LIN {X 98.42, Y 171.93, Z 0.00, A 0, B 0, C 0} C_DIS
LIN {X 98.57, Y 172.17, Z 0.00, A 0, B 0, C 0} C_DIS
LIN {X 98.70, Y 172.42, Z 0.00, A 0, B 0, C 0} C_DIS
LIN {X 98.83, Y 172.69, Z 0.00, A 0, B 0, C 0} C_DIS
LIN {X 98.95, Y 172.96, Z 0.00, A 0, B 0, C 0} C_DIS
LIN {X 99.07, Y 173.23, Z 0.00, A 0, B 0, C 0} C_DIS
LIN {X 99.19, Y 173.50, Z 0.00, A 0, B 0, C 0} C_DIS
LIN {X 99.31, Y 173.78, Z 0.00, A 0, B 0, C 0} C_DIS
LIN {X 99.43, Y 174.05, Z 0.00, A 0, B 0, C 0} C_DIS
LIN {X 99.55, Y 174.33, Z 0.00, A 0, B 0, C 0} C_DIS
LIN {X 99.67, Y 174.60, Z 0.00, A 0, B 0, C 0} C_DIS
LIN {X 99.79, Y 174.87, Z 0.00, A 0, B 0, C 0} C_DIS
LIN {X 99.92, Y 175.14, Z 0.00, A 0, B 0, C 0} C_DIS
LIN {X 100.03, Y 175.42, Z 0.00, A 0, B 0, C 0} C_DIS
LIN {X 100.12, Y 175.71, Z 0.00, A 0, B 0, C 0} C_DIS
LIN {X 100.21, Y 176.02, Z 0.00, A 0, B 0, C 0} C_DIS
LIN {X 100.30, Y 176.31, Z 0.00, A 0, B 0, C 0} C_DIS
LIN {X 100.41, Y 176.59, Z 0.00, A 0, B 0, C 0} C_DIS
LIN {X 100.52, Y 176.87, Z 0.00, A 0, B 0, C 0} C_DIS
LIN {X 100.64, Y 177.14, Z 0.00, A 0, B 0, C 0} C_DIS
LIN {X 100.77, Y 177.41, Z 0.00, A 0, B 0, C 0} C_DIS
LIN {X 100.89, Y 177.68, Z 0.00, A 0, B 0, C 0} C_DIS
LIN {X 101.02, Y 177.95, Z 0.00, A 0, B 0, C 0} C_DIS
LIN {X 101.14, Y 178.22, Z 0.00, A 0, B 0, C 0} C_DIS
LIN {X 101.26, Y 178.50, Z 0.00, A 0, B 0, C 0} C_DIS
LIN {X 101.36, Y 178.79, Z 0.00, A 0, B 0, C 0} C_DIS
LIN {X 101.45, Y 179.08, Z 0.00, A 0, B 0, C 0} C_DIS
LIN {X 101.54, Y 179.38, Z 0.00, A 0, B 0, C 0} C_DIS
LIN {X 101.64, Y 179.67, Z 0.00, A 0, B 0, C 0} C_DIS
LIN {X 101.75, Y 179.95, Z 0.00, A 0, B 0, C 0} C_DIS
LIN {X 101.85, Y 180.24, Z 0.00, A 0, B 0, C 0} C_DIS
LIN {X 101.93, Y 180.55, Z 0.00, A 0, B 0, C 0} C_DIS
LIN {X 102.02, Y 180.85, Z 0.00, A 0, B 0, C 0} C_DIS
LIN {X 102.12, Y 181.13, Z 0.00, A 0, B 0, C 0} C_DIS
LIN {X 102.23, Y 181.41, Z 0.00, A 0, B 0, C 0} C_DIS
LIN {X 102.33, Y 181.71, Z 0.00, A 0, B 0, C 0} C_DIS
LIN {X 102.41, Y 182.01, Z 0.00, A 0, B 0, C 0} C_DIS
LIN {X 102.51, Y 182.30, Z 0.00, A 0, B 0, C 0} C_DIS
LIN {X 102.61, Y 182.59, Z 0.00, A 0, B 0, C 0} C_DIS
LIN {X 102.72, Y 182.87, Z 0.00, A 0, B 0, C 0} C_DIS
LIN {X 102.81, Y 183.17, Z 0.00, A 0, B 0, C 0} C_DIS
LIN {X 102.89, Y 183.48, Z 0.00, A 0, B 0, C 0} C_DIS
LIN {X 103.00, Y 183.76, Z 0.00, A 0, B 0, C 0} C_DIS
LIN {X 103.12, Y 184.03, Z 0.00, A 0, B 0, C 0} C_DIS
LIN {X 103.20, Y 184.34, Z 0.00, A 0, B 0, C 0} C_DIS
LIN {X 103.25, Y 184.65, Z 0.00, A 0, B 0, C 0} C_DIS
LIN {X 103.31, Y 184.97, Z 0.00, A 0, B 0, C 0} C_DIS
LIN {X 103.40, Y 185.27, Z 0.00, A 0, B 0, C 0} C_DIS
LIN {X 103.49, Y 185.57, Z 0.00, A 0, B 0, C 0} C_DIS
LIN {X 103.57, Y 185.87, Z 0.00, A 0, B 0, C 0} C_DIS
LIN {X 103.62, Y 186.19, Z 0.00, A 0, B 0, C 0} C_DIS
LIN {X 103.67, Y 186.51, Z 0.00, A 0, B 0, C 0} C_DIS
LIN {X 103.72, Y 186.83, Z 0.00, A 0, B 0, C 0} C_DIS
LIN {X 103.80, Y 187.13, Z 0.00, A 0, B 0, C 0} C_DIS
LIN {X 103.89, Y 187.43, Z 0.00, A 0, B 0, C 0} C_DIS
LIN {X 103.98, Y 187.73, Z 0.00, A 0, B 0, C 0} C_DIS
LIN {X 104.04, Y 188.04, Z 0.00, A 0, B 0, C 0} C_DIS
LIN {X 104.09, Y 188.37, Z 0.00, A 0, B 0, C 0} C_DIS
LIN {X 104.13, Y 188.69, Z 0.00, A 0, B 0, C 0} C_DIS
LIN {X 104.21, Y 189.00, Z 0.00, A 0, B 0, C 0} C_DIS
LIN {X 104.30, Y 189.29, Z 0.00, A 0, B 0, C 0} C_DIS
LIN {X 104.38, Y 189.59, Z 0.00, A 0, B 0, C 0} C_DIS
LIN {X 104.45, Y 189.91, Z 0.00, A 0, B 0, C 0} C_DIS
LIN {X 104.51, Y 190.22, Z 0.00, A 0, B 0, C 0} C_DIS
LIN {X 104.56, Y 190.54, Z 0.00, A 0, B 0, C 0} C_DIS
LIN {X 104.62, Y 190.85, Z 0.00, A 0, B 0, C 0} C_DIS
LIN {X 104.70, Y 191.16, Z 0.00, A 0, B 0, C 0} C_DIS
LIN {X 104.78, Y 191.46, Z 0.00, A 0, B 0, C 0} C_DIS
LIN {X 104.86, Y 191.77, Z 0.00, A 0, B 0, C 0} C_DIS
LIN {X 104.93, Y 192.08, Z 0.00, A 0, B 0, C 0} C_DIS
LIN {X 104.99, Y 192.39, Z 0.00, A 0, B 0, C 0} C_DIS
LIN {X 105.04, Y 192.71, Z 0.00, A 0, B 0, C 0} C_DIS
LIN {X 105.08, Y 193.03, Z 0.00, A 0, B 0, C 0} C_DIS
LIN {X 105.13, Y 193.35, Z 0.00, A 0, B 0, C 0} C_DIS
LIN {X 105.18, Y 193.67, Z 0.00, A 0, B 0, C 0} C_DIS
LIN {X 105.23, Y 193.99, Z 0.00, A 0, B 0, C 0} C_DIS
LIN {X 105.29, Y 194.31, Z 0.00, A 0, B 0, C 0} C_DIS
LIN {X 105.35, Y 194.62, Z 0.00, A 0, B 0, C 0} C_DIS
LIN {X 105.41, Y 194.94, Z 0.00, A 0, B 0, C 0} C_DIS
LIN {X 105.46, Y 195.25, Z 0.00, A 0, B 0, C 0} C_DIS
LIN {X 105.50, Y 195.57, Z 0.00, A 0, B 0, C 0} C_DIS
LIN {X 105.54, Y 195.90, Z 0.00, A 0, B 0, C 0} C_DIS
LIN {X 105.58, Y 196.22, Z 0.00, A 0, B 0, C 0} C_DIS
LIN {X 105.61, Y 196.54, Z 0.00, A 0, B 0, C 0} C_DIS
LIN {X 105.64, Y 196.87, Z 0.00, A 0, B 0, C 0} C_DIS
LIN {X 105.67, Y 197.19, Z 0.00, A 0, B 0, C 0} C_DIS
LIN {X 105.71, Y 197.51, Z 0.00, A 0, B 0, C 0} C_DIS
LIN {X 105.76, Y 197.83, Z 0.00, A 0, B 0, C 0} C_DIS
LIN {X 105.82, Y 198.15, Z 0.00, A 0, B 0, C 0} C_DIS
LIN {X 105.88, Y 198.46, Z 0.00, A 0, B 0, C 0} C_DIS
LIN {X 105.93, Y 198.78, Z 0.00, A 0, B 0, C 0} C_DIS
LIN {X 105.98, Y 199.10, Z 0.00, A 0, B 0, C 0} C_DIS
LIN {X 106.02, Y 199.42, Z 0.00, A 0, B 0, C 0} C_DIS
LIN {X 106.04, Y 199.75, Z 0.00, A 0, B 0, C 0} C_DIS
LIN {X 106.04, Y 200.08, Z 0.00, A 0, B 0, C 0} C_DIS
LIN {X 106.04, Y 200.41, Z 0.00, A 0, B 0, C 0} C_DIS
LIN {X 106.03, Y 200.74, Z 0.00, A 0, B 0, C 0} C_DIS
LIN {X 106.03, Y 201.06, Z 0.00, A 0, B 0, C 0} C_DIS
LIN {X 106.05, Y 201.39, Z 0.00, A 0, B 0, C 0} C_DIS
LIN {X 106.09, Y 201.71, Z 0.00, A 0, B 0, C 0} C_DIS
LIN {X 106.13, Y 202.03, Z 0.00, A 0, B 0, C 0} C_DIS
LIN {X 106.19, Y 202.35, Z 0.00, A 0, B 0, C 0} C_DIS
LIN {X 106.25, Y 202.66, Z 0.00, A 0, B 0, C 0} C_DIS
LIN {X 106.30, Y 202.98, Z 0.00, A 0, B 0, C 0} C_DIS
LIN {X 106.36, Y 203.30, Z 0.00, A 0, B 0, C 0} C_DIS
LIN {X 106.40, Y 203.62, Z 0.00, A 0, B 0, C 0} C_DIS
LIN {X 106.43, Y 203.94, Z 0.00, A 0, B 0, C 0} C_DIS
LIN {X 106.46, Y 204.27, Z 0.00, A 0, B 0, C 0} C_DIS
LIN {X 106.48, Y 204.59, Z 0.00, A 0, B 0, C 0} C_DIS
LIN {X 106.48, Y 204.92, Z 0.00, A 0, B 0, C 0} C_DIS
LIN {X 106.48, Y 205.25, Z 0.00, A 0, B 0, C 0} C_DIS
LIN {X 106.47, Y 205.58, Z 0.00, A 0, B 0, C 0} C_DIS
LIN {X 106.46, Y 205.91, Z 0.00, A 0, B 0, C 0} C_DIS
LIN {X 106.46, Y 206.24, Z 0.00, A 0, B 0, C 0} C_DIS
LIN {X 106.48, Y 206.56, Z 0.00, A 0, B 0, C 0} C_DIS
LIN {X 106.52, Y 206.88, Z 0.00, A 0, B 0, C 0} C_DIS
LIN {X 106.56, Y 207.20, Z 0.00, A 0, B 0, C 0} C_DIS
LIN {X 106.61, Y 207.52, Z 0.00, A 0, B 0, C 0} C_DIS
LIN {X 106.66, Y 207.85, Z 0.00, A 0, B 0, C 0} C_DIS
LIN {X 106.73, Y 208.16, Z 0.00, A 0, B 0, C 0} C_DIS
LIN {X 106.83, Y 208.44, Z 0.00, A 0, B 0, C 0} C_DIS
LIN {X 106.96, Y 208.69, Z 0.00, A 0, B 0, C 0} C_DIS
LIN {X 107.12, Y 208.92, Z 0.00, A 0, B 0, C 0} C_DIS
LIN {X 107.28, Y 209.15, Z 0.00, A 0, B 0, C 0} C_DIS
LIN {X 107.43, Y 209.39, Z 0.00, A 0, B 0, C 0} C_DIS
LIN {X 107.60, Y 209.58, Z 0.00, A 0, B 0, C 0} C_DIS
LIN {X 107.80, Y 209.69, Z 0.00, A 0, B 0, C 0} C_DIS
LIN {X 108.02, Y 209.75, Z 0.00, A 0, B 0, C 0} C_DIS
LIN {X 108.24, Y 209.76, Z 0.00, A 0, B 0, C 0} C_DIS
LIN {X 108.46, Y 209.74, Z 0.00, A 0, B 0, C 0} C_DIS
LIN {X 108.67, Y 209.69, Z 0.00, A 0, B 0, C 0} C_DIS
LIN {X 108.89, Y 209.62, Z 0.00, A 0, B 0, C 0} C_DIS
LIN {X 109.10, Y 209.55, Z 0.00, A 0, B 0, C 0} C_DIS
LIN {X 109.31, Y 209.46, Z 0.00, A 0, B 0, C 0} C_DIS
LIN {X 109.52, Y 209.38, Z 0.00, A 0, B 0, C 0} C_DIS
LIN {X 109.73, Y 209.30, Z 0.00, A 0, B 0, C 0} C_DIS
LIN {X 109.94, Y 209.23, Z 0.00, A 0, B 0, C 0} C_DIS
LIN {X 110.15, Y 209.15, Z 0.00, A 0, B 0, C 0} C_DIS
LIN {X 110.36, Y 209.07, Z 0.00, A 0, B 0, C 0} C_DIS
LIN {X 110.57, Y 208.98, Z 0.00, A 0, B 0, C 0} C_DIS
LIN {X 110.78, Y 208.89, Z 0.00, A 0, B 0, C 0} C_DIS
LIN {X 111.00, Y 208.82, Z 0.00, A 0, B 0, C 0} C_DIS
LIN {X 111.21, Y 208.76, Z 0.00, A 0, B 0, C 0} C_DIS
LIN {X 111.42, Y 208.73, Z 0.00, A 0, B 0, C 0} C_DIS
LIN {X 111.64, Y 208.72, Z 0.00, A 0, B 0, C 0} C_DIS
LIN {X 111.86, Y 208.72, Z 0.00, A 0, B 0, C 0} C_DIS
LIN {X 112.08, Y 208.72, Z 0.00, A 0, B 0, C 0} C_DIS
LIN {X 112.29, Y 208.72, Z 0.00, A 0, B 0, C 0} C_DIS
LIN {X 112.51, Y 208.72, Z 0.00, A 0, B 0, C 0} C_DIS
LIN {X 112.73, Y 208.72, Z 0.00, A 0, B 0, C 0} C_DIS
LIN {X 112.95, Y 208.72, Z 0.00, A 0, B 0, C 0} C_DIS
LIN {X 113.16, Y 208.72, Z 0.00, A 0, B 0, C 0} C_DIS
LIN {X 113.38, Y 208.72, Z 0.00, A 0, B 0, C 0} C_DIS
LIN {X 113.60, Y 208.72, Z 0.00, A 0, B 0, C 0} C_DIS
LIN {X 113.82, Y 208.72, Z 0.00, A 0, B 0, C 0} C_DIS
LIN {X 114.03, Y 208.72, Z 0.00, A 0, B 0, C 0} C_DIS
LIN {X 114.25, Y 208.72, Z 0.00, A 0, B 0, C 0} C_DIS
LIN {X 114.47, Y 208.72, Z 0.00, A 0, B 0, C 0} C_DIS
LIN {X 114.69, Y 208.72, Z 0.00, A 0, B 0, C 0} C_DIS
LIN {X 114.90, Y 208.73, Z 0.00, A 0, B 0, C 0} C_DIS
LIN {X 115.12, Y 208.73, Z 0.00, A 0, B 0, C 0} C_DIS
LIN {X 115.34, Y 208.73, Z 0.00, A 0, B 0, C 0} C_DIS
LIN {X 115.56, Y 208.73, Z 0.00, A 0, B 0, C 0} C_DIS
LIN {X 115.77, Y 208.73, Z 0.00, A 0, B 0, C 0} C_DIS
LIN {X 115.99, Y 208.73, Z 0.00, A 0, B 0, C 0} C_DIS
LIN {X 116.21, Y 208.72, Z 0.00, A 0, B 0, C 0} C_DIS
LIN {X 116.43, Y 208.72, Z 0.00, A 0, B 0, C 0} C_DIS
LIN {X 116.64, Y 208.72, Z 0.00, A 0, B 0, C 0} C_DIS
LIN {X 116.86, Y 208.72, Z 0.00, A 0, B 0, C 0} C_DIS
LIN {X 117.08, Y 208.72, Z 0.00, A 0, B 0, C 0} C_DIS
LIN {X 117.30, Y 208.72, Z 0.00, A 0, B 0, C 0} C_DIS
LIN {X 117.51, Y 208.72, Z 0.00, A 0, B 0, C 0} C_DIS
LIN {X 117.73, Y 208.72, Z 0.00, A 0, B 0, C 0} C_DIS
LIN {X 117.95, Y 208.72, Z 0.00, A 0, B 0, C 0} C_DIS
LIN {X 118.17, Y 208.72, Z 0.00, A 0, B 0, C 0} C_DIS
LIN {X 118.38, Y 208.72, Z 0.00, A 0, B 0, C 0} C_DIS
LIN {X 118.60, Y 208.73, Z 0.00, A 0, B 0, C 0} C_DIS
LIN {X 118.82, Y 208.73, Z 0.00, A 0, B 0, C 0} C_DIS
LIN {X 119.04, Y 208.74, Z 0.00, A 0, B 0, C 0} C_DIS
LIN {X 119.25, Y 208.74, Z 0.00, A 0, B 0, C 0} C_DIS
LIN {X 119.47, Y 208.73, Z 0.00, A 0, B 0, C 0} C_DIS
LIN {X 119.69, Y 208.72, Z 0.00, A 0, B 0, C 0} C_DIS
LIN {X 119.90, Y 208.69, Z 0.00, A 0, B 0, C 0} C_DIS
LIN {X 120.12, Y 208.65, Z 0.00, A 0, B 0, C 0} C_DIS
LIN {X 120.33, Y 208.59, Z 0.00, A 0, B 0, C 0} C_DIS
LIN {X 120.55, Y 208.52, Z 0.00, A 0, B 0, C 0} C_DIS
LIN {X 120.76, Y 208.44, Z 0.00, A 0, B 0, C 0} C_DIS
LIN {X 120.96, Y 208.33, Z 0.00, A 0, B 0, C 0} C_DIS
LIN {X 121.16, Y 208.19, Z 0.00, A 0, B 0, C 0} C_DIS
LIN {X 121.32, Y 207.98, Z 0.00, A 0, B 0, C 0} C_DIS
LIN {X 121.47, Y 207.75, Z 0.00, A 0, B 0, C 0} C_DIS
LIN {X 121.64, Y 207.52, Z 0.00, A 0, B 0, C 0} C_DIS
LIN {X 121.78, Y 207.28, Z 0.00, A 0, B 0, C 0} C_DIS
LIN {X 121.90, Y 207.01, Z 0.00, A 0, B 0, C 0} C_DIS
LIN {X 121.99, Y 206.71, Z 0.00, A 0, B 0, C 0} C_DIS
LIN {X 122.06, Y 206.40, Z 0.00, A 0, B 0, C 0} C_DIS
LIN {X 122.11, Y 206.08, Z 0.00, A 0, B 0, C 0} C_DIS
LIN {X 122.15, Y 205.76, Z 0.00, A 0, B 0, C 0} C_DIS
LIN {X 122.17, Y 205.43, Z 0.00, A 0, B 0, C 0} C_DIS
LIN {X 122.20, Y 205.11, Z 0.00, A 0, B 0, C 0} C_DIS
LIN {X 122.21, Y 204.78, Z 0.00, A 0, B 0, C 0} C_DIS
LIN {X 122.22, Y 204.45, Z 0.00, A 0, B 0, C 0} C_DIS
LIN {X 122.22, Y 204.13, Z 0.00, A 0, B 0, C 0} C_DIS
LIN {X 122.22, Y 203.80, Z 0.00, A 0, B 0, C 0} C_DIS
LIN {X 122.22, Y 203.47, Z 0.00, A 0, B 0, C 0} C_DIS
LIN {X 122.22, Y 203.14, Z 0.00, A 0, B 0, C 0} C_DIS
LIN {X 122.22, Y 202.82, Z 0.00, A 0, B 0, C 0} C_DIS
LIN {X 122.21, Y 202.49, Z 0.00, A 0, B 0, C 0} C_DIS
LIN {X 122.21, Y 202.16, Z 0.00, A 0, B 0, C 0} C_DIS
LIN {X 122.21, Y 201.83, Z 0.00, A 0, B 0, C 0} C_DIS
LIN {X 122.21, Y 201.51, Z 0.00, A 0, B 0, C 0} C_DIS
LIN {X 122.21, Y 201.18, Z 0.00, A 0, B 0, C 0} C_DIS
LIN {X 122.21, Y 200.85, Z 0.00, A 0, B 0, C 0} C_DIS
LIN {X 122.21, Y 200.52, Z 0.00, A 0, B 0, C 0} C_DIS
LIN {X 122.22, Y 200.20, Z 0.00, A 0, B 0, C 0} C_DIS
LIN {X 122.22, Y 199.87, Z 0.00, A 0, B 0, C 0} C_DIS
LIN {X 122.22, Y 199.54, Z 0.00, A 0, B 0, C 0} C_DIS
LIN {X 122.22, Y 199.21, Z 0.00, A 0, B 0, C 0} C_DIS
LIN {X 122.22, Y 198.88, Z 0.00, A 0, B 0, C 0} C_DIS
LIN {X 122.22, Y 198.56, Z 0.00, A 0, B 0, C 0} C_DIS
LIN {X 122.20, Y 198.23, Z 0.00, A 0, B 0, C 0} C_DIS
LIN {X 122.20, Y 197.90, Z 0.00, A 0, B 0, C 0} C_DIS
LIN {X 122.21, Y 197.58, Z 0.00, A 0, B 0, C 0} C_DIS
LIN {X 122.25, Y 197.25, Z 0.00, A 0, B 0, C 0} C_DIS
LIN {X 122.34, Y 196.94, Z 0.00, A 0, B 0, C 0} C_DIS
LIN {X 122.46, Y 196.66, Z 0.00, A 0, B 0, C 0} C_DIS
LIN {X 122.62, Y 196.45, Z 0.00, A 0, B 0, C 0} C_DIS
LIN {X 122.82, Y 196.34, Z 0.00, A 0, B 0, C 0} C_DIS
LIN {X 123.03, Y 196.30, Z 0.00, A 0, B 0, C 0} C_DIS
LIN {X 123.25, Y 196.28, Z 0.00, A 0, B 0, C 0} C_DIS
LIN {X 123.47, Y 196.28, Z 0.00, A 0, B 0, C 0} C_DIS
LIN {X 123.69, Y 196.27, Z 0.00, A 0, B 0, C 0} C_DIS
LIN {X 123.91, Y 196.27, Z 0.00, A 0, B 0, C 0} C_DIS
LIN {X 124.13, Y 196.27, Z 0.00, A 0, B 0, C 0} C_DIS
LIN {X 124.35, Y 196.27, Z 0.00, A 0, B 0, C 0} C_DIS
LIN {X 124.56, Y 196.26, Z 0.00, A 0, B 0, C 0} C_DIS
LIN {X 124.78, Y 196.26, Z 0.00, A 0, B 0, C 0} C_DIS
LIN {X 125.00, Y 196.26, Z 0.00, A 0, B 0, C 0} C_DIS
LIN {X 125.22, Y 196.27, Z 0.00, A 0, B 0, C 0} C_DIS
LIN {X 125.43, Y 196.27, Z 0.00, A 0, B 0, C 0} C_DIS
LIN {X 125.65, Y 196.27, Z 0.00, A 0, B 0, C 0} C_DIS
LIN {X 125.87, Y 196.27, Z 0.00, A 0, B 0, C 0} C_DIS
LIN {X 126.08, Y 196.27, Z 0.00, A 0, B 0, C 0} C_DIS
LIN {X 126.30, Y 196.27, Z 0.00, A 0, B 0, C 0} C_DIS
LIN {X 126.52, Y 196.27, Z 0.00, A 0, B 0, C 0} C_DIS
LIN {X 126.73, Y 196.27, Z 0.00, A 0, B 0, C 0} C_DIS
LIN {X 126.95, Y 196.27, Z 0.00, A 0, B 0, C 0} C_DIS
LIN {X 127.17, Y 196.27, Z 0.00, A 0, B 0, C 0} C_DIS
LIN {X 127.39, Y 196.27, Z 0.00, A 0, B 0, C 0} C_DIS
LIN {X 127.60, Y 196.27, Z 0.00, A 0, B 0, C 0} C_DIS
LIN {X 127.82, Y 196.27, Z 0.00, A 0, B 0, C 0} C_DIS
LIN {X 128.04, Y 196.27, Z 0.00, A 0, B 0, C 0} C_DIS
LIN {X 128.26, Y 196.27, Z 0.00, A 0, B 0, C 0} C_DIS
LIN {X 128.48, Y 196.27, Z 0.00, A 0, B 0, C 0} C_DIS
LIN {X 128.69, Y 196.27, Z 0.00, A 0, B 0, C 0} C_DIS
LIN {X 128.91, Y 196.27, Z 0.00, A 0, B 0, C 0} C_DIS
LIN {X 129.13, Y 196.27, Z 0.00, A 0, B 0, C 0} C_DIS
LIN {X 129.34, Y 196.28, Z 0.00, A 0, B 0, C 0} C_DIS
LIN {X 129.56, Y 196.28, Z 0.00, A 0, B 0, C 0} C_DIS
LIN {X 129.78, Y 196.27, Z 0.00, A 0, B 0, C 0} C_DIS
LIN {X 130.00, Y 196.26, Z 0.00, A 0, B 0, C 0} C_DIS
LIN {X 130.21, Y 196.26, Z 0.00, A 0, B 0, C 0} C_DIS
LIN {X 130.43, Y 196.28, Z 0.00, A 0, B 0, C 0} C_DIS
LIN {X 130.65, Y 196.35, Z 0.00, A 0, B 0, C 0} C_DIS
LIN {X 130.85, Y 196.47, Z 0.00, A 0, B 0, C 0} C_DIS
LIN {X 131.02, Y 196.66, Z 0.00, A 0, B 0, C 0} C_DIS
LIN {X 131.15, Y 196.92, Z 0.00, A 0, B 0, C 0} C_DIS
LIN {X 131.21, Y 197.24, Z 0.00, A 0, B 0, C 0} C_DIS
LIN {X 131.25, Y 197.57, Z 0.00, A 0, B 0, C 0} C_DIS
LIN {X 131.27, Y 197.89, Z 0.00, A 0, B 0, C 0} C_DIS
LIN {X 131.27, Y 198.22, Z 0.00, A 0, B 0, C 0} C_DIS
LIN {X 131.27, Y 198.55, Z 0.00, A 0, B 0, C 0} C_DIS
LIN {X 131.26, Y 198.88, Z 0.00, A 0, B 0, C 0} C_DIS
LIN {X 131.26, Y 199.20, Z 0.00, A 0, B 0, C 0} C_DIS
LIN {X 131.26, Y 199.53, Z 0.00, A 0, B 0, C 0} C_DIS
LIN {X 131.26, Y 199.86, Z 0.00, A 0, B 0, C 0} C_DIS
LIN {X 131.26, Y 200.19, Z 0.00, A 0, B 0, C 0} C_DIS
LIN {X 131.26, Y 200.51, Z 0.00, A 0, B 0, C 0} C_DIS
LIN {X 131.26, Y 200.84, Z 0.00, A 0, B 0, C 0} C_DIS
LIN {X 131.26, Y 201.17, Z 0.00, A 0, B 0, C 0} C_DIS
LIN {X 131.26, Y 201.50, Z 0.00, A 0, B 0, C 0} C_DIS
LIN {X 131.26, Y 201.83, Z 0.00, A 0, B 0, C 0} C_DIS
LIN {X 131.26, Y 202.15, Z 0.00, A 0, B 0, C 0} C_DIS
LIN {X 131.26, Y 202.48, Z 0.00, A 0, B 0, C 0} C_DIS
LIN {X 131.26, Y 202.81, Z 0.00, A 0, B 0, C 0} C_DIS
LIN {X 131.26, Y 203.14, Z 0.00, A 0, B 0, C 0} C_DIS
LIN {X 131.26, Y 203.46, Z 0.00, A 0, B 0, C 0} C_DIS
LIN {X 131.26, Y 203.79, Z 0.00, A 0, B 0, C 0} C_DIS
LIN {X 131.26, Y 204.12, Z 0.00, A 0, B 0, C 0} C_DIS
LIN {X 131.26, Y 204.45, Z 0.00, A 0, B 0, C 0} C_DIS
LIN {X 131.26, Y 204.77, Z 0.00, A 0, B 0, C 0} C_DIS
LIN {X 131.26, Y 205.10, Z 0.00, A 0, B 0, C 0} C_DIS
LIN {X 131.26, Y 205.43, Z 0.00, A 0, B 0, C 0} C_DIS
LIN {X 131.26, Y 205.76, Z 0.00, A 0, B 0, C 0} C_DIS
LIN {X 131.26, Y 206.09, Z 0.00, A 0, B 0, C 0} C_DIS
LIN {X 131.26, Y 206.41, Z 0.00, A 0, B 0, C 0} C_DIS
LIN {X 131.26, Y 206.74, Z 0.00, A 0, B 0, C 0} C_DIS
LIN {X 131.26, Y 207.07, Z 0.00, A 0, B 0, C 0} C_DIS
LIN {X 131.26, Y 207.40, Z 0.00, A 0, B 0, C 0} C_DIS
LIN {X 131.26, Y 207.72, Z 0.00, A 0, B 0, C 0} C_DIS
LIN {X 131.26, Y 208.05, Z 0.00, A 0, B 0, C 0} C_DIS
LIN {X 131.26, Y 208.38, Z 0.00, A 0, B 0, C 0} C_DIS
LIN {X 131.26, Y 208.71, Z 0.00, A 0, B 0, C 0} C_DIS
LIN {X 131.26, Y 209.04, Z 0.00, A 0, B 0, C 0} C_DIS
LIN {X 131.26, Y 209.36, Z 0.00, A 0, B 0, C 0} C_DIS
LIN {X 131.26, Y 209.69, Z 0.00, A 0, B 0, C 0} C_DIS
LIN {X 131.26, Y 210.02, Z 0.00, A 0, B 0, C 0} C_DIS
LIN {X 131.26, Y 210.35, Z 0.00, A 0, B 0, C 0} C_DIS
LIN {X 131.26, Y 210.67, Z 0.00, A 0, B 0, C 0} C_DIS
LIN {X 131.26, Y 211.00, Z 0.00, A 0, B 0, C 0} C_DIS
LIN {X 131.26, Y 211.33, Z 0.00, A 0, B 0, C 0} C_DIS
LIN {X 131.26, Y 211.66, Z 0.00, A 0, B 0, C 0} C_DIS
LIN {X 131.26, Y 211.98, Z 0.00, A 0, B 0, C 0} C_DIS
LIN {X 131.26, Y 212.31, Z 0.00, A 0, B 0, C 0} C_DIS
LIN {X 131.26, Y 212.64, Z 0.00, A 0, B 0, C 0} C_DIS
LIN {X 131.26, Y 212.97, Z 0.00, A 0, B 0, C 0} C_DIS
LIN {X 131.26, Y 213.30, Z 0.00, A 0, B 0, C 0} C_DIS
LIN {X 131.26, Y 213.62, Z 0.00, A 0, B 0, C 0} C_DIS
LIN {X 131.26, Y 213.95, Z 0.00, A 0, B 0, C 0} C_DIS
LIN {X 131.26, Y 214.28, Z 0.00, A 0, B 0, C 0} C_DIS
LIN {X 131.26, Y 214.61, Z 0.00, A 0, B 0, C 0} C_DIS
LIN {X 131.26, Y 214.93, Z 0.00, A 0, B 0, C 0} C_DIS
LIN {X 131.26, Y 215.26, Z 0.00, A 0, B 0, C 0} C_DIS
LIN {X 131.26, Y 215.59, Z 0.00, A 0, B 0, C 0} C_DIS
LIN {X 131.26, Y 215.92, Z 0.00, A 0, B 0, C 0} C_DIS
LIN {X 131.26, Y 216.24, Z 0.00, A 0, B 0, C 0} C_DIS
LIN {X 131.26, Y 216.57, Z 0.00, A 0, B 0, C 0} C_DIS
LIN {X 131.26, Y 216.90, Z 0.00, A 0, B 0, C 0} C_DIS
LIN {X 131.26, Y 217.23, Z 0.00, A 0, B 0, C 0} C_DIS
LIN {X 131.26, Y 217.56, Z 0.00, A 0, B 0, C 0} C_DIS
LIN {X 131.26, Y 217.88, Z 0.00, A 0, B 0, C 0} C_DIS
LIN {X 131.26, Y 218.21, Z 0.00, A 0, B 0, C 0} C_DIS
LIN {X 131.26, Y 218.54, Z 0.00, A 0, B 0, C 0} C_DIS
LIN {X 131.26, Y 218.87, Z 0.00, A 0, B 0, C 0} C_DIS
LIN {X 131.26, Y 219.19, Z 0.00, A 0, B 0, C 0} C_DIS
LIN {X 131.26, Y 219.52, Z 0.00, A 0, B 0, C 0} C_DIS
LIN {X 131.26, Y 219.85, Z 0.00, A 0, B 0, C 0} C_DIS
LIN {X 131.26, Y 220.18, Z 0.00, A 0, B 0, C 0} C_DIS
LIN {X 131.26, Y 220.51, Z 0.00, A 0, B 0, C 0} C_DIS
LIN {X 131.26, Y 220.83, Z 0.00, A 0, B 0, C 0} C_DIS
LIN {X 131.26, Y 221.16, Z 0.00, A 0, B 0, C 0} C_DIS
LIN {X 131.26, Y 221.49, Z 0.00, A 0, B 0, C 0} C_DIS
LIN {X 131.26, Y 221.82, Z 0.00, A 0, B 0, C 0} C_DIS
LIN {X 131.26, Y 222.14, Z 0.00, A 0, B 0, C 0} C_DIS
LIN {X 131.26, Y 222.47, Z 0.00, A 0, B 0, C 0} C_DIS
LIN {X 131.26, Y 222.80, Z 0.00, A 0, B 0, C 0} C_DIS
LIN {X 131.26, Y 223.13, Z 0.00, A 0, B 0, C 0} C_DIS
LIN {X 131.26, Y 223.45, Z 0.00, A 0, B 0, C 0} C_DIS
LIN {X 131.26, Y 223.78, Z 0.00, A 0, B 0, C 0} C_DIS
LIN {X 131.26, Y 224.11, Z 0.00, A 0, B 0, C 0} C_DIS
LIN {X 131.26, Y 224.44, Z 0.00, A 0, B 0, C 0} C_DIS
LIN {X 131.26, Y 224.77, Z 0.00, A 0, B 0, C 0} C_DIS
LIN {X 131.26, Y 225.09, Z 0.00, A 0, B 0, C 0} C_DIS
LIN {X 131.26, Y 225.42, Z 0.00, A 0, B 0, C 0} C_DIS
LIN {X 131.26, Y 225.75, Z 0.00, A 0, B 0, C 0} C_DIS
LIN {X 131.26, Y 226.08, Z 0.00, A 0, B 0, C 0} C_DIS
LIN {X 131.26, Y 226.40, Z 0.00, A 0, B 0, C 0} C_DIS
LIN {X 131.26, Y 226.73, Z 0.00, A 0, B 0, C 0} C_DIS
LIN {X 131.26, Y 227.06, Z 0.00, A 0, B 0, C 0} C_DIS
LIN {X 131.26, Y 227.39, Z 0.00, A 0, B 0, C 0} C_DIS
LIN {X 131.26, Y 227.71, Z 0.00, A 0, B 0, C 0} C_DIS
LIN {X 131.26, Y 228.04, Z 0.00, A 0, B 0, C 0} C_DIS
LIN {X 131.26, Y 228.37, Z 0.00, A 0, B 0, C 0} C_DIS
LIN {X 131.26, Y 228.70, Z 0.00, A 0, B 0, C 0} C_DIS
LIN {X 131.26, Y 229.03, Z 0.00, A 0, B 0, C 0} C_DIS
LIN {X 131.26, Y 229.35, Z 0.00, A 0, B 0, C 0} C_DIS
LIN {X 131.26, Y 229.68, Z 0.00, A 0, B 0, C 0} C_DIS
LIN {X 131.26, Y 230.01, Z 0.00, A 0, B 0, C 0} C_DIS
LIN {X 131.26, Y 230.34, Z 0.00, A 0, B 0, C 0} C_DIS
LIN {X 131.26, Y 230.66, Z 0.00, A 0, B 0, C 0} C_DIS
LIN {X 131.26, Y 230.99, Z 0.00, A 0, B 0, C 0} C_DIS
LIN {X 131.26, Y 231.32, Z 0.00, A 0, B 0, C 0} C_DIS
LIN {X 131.26, Y 231.65, Z 0.00, A 0, B 0, C 0} C_DIS
LIN {X 131.26, Y 231.98, Z 0.00, A 0, B 0, C 0} C_DIS
LIN {X 131.26, Y 232.30, Z 0.00, A 0, B 0, C 0} C_DIS
LIN {X 131.26, Y 232.63, Z 0.00, A 0, B 0, C 0} C_DIS
LIN {X 131.26, Y 232.96, Z 0.00, A 0, B 0, C 0} C_DIS
LIN {X 131.26, Y 233.29, Z 0.00, A 0, B 0, C 0} C_DIS
LIN {X 131.26, Y 233.61, Z 0.00, A 0, B 0, C 0} C_DIS
LIN {X 131.26, Y 233.94, Z 0.00, A 0, B 0, C 0} C_DIS
LIN {X 131.26, Y 234.27, Z 0.00, A 0, B 0, C 0} C_DIS
LIN {X 131.26, Y 234.60, Z 0.00, A 0, B 0, C 0} C_DIS
LIN {X 131.26, Y 234.92, Z 0.00, A 0, B 0, C 0} C_DIS
LIN {X 131.26, Y 235.25, Z 0.00, A 0, B 0, C 0} C_DIS
LIN {X 131.26, Y 235.58, Z 0.00, A 0, B 0, C 0} C_DIS
LIN {X 131.26, Y 235.91, Z 0.00, A 0, B 0, C 0} C_DIS
LIN {X 131.26, Y 236.24, Z 0.00, A 0, B 0, C 0} C_DIS
LIN {X 131.26, Y 236.56, Z 0.00, A 0, B 0, C 0} C_DIS
LIN {X 131.26, Y 236.89, Z 0.00, A 0, B 0, C 0} C_DIS
LIN {X 131.26, Y 237.22, Z 0.00, A 0, B 0, C 0} C_DIS
LIN {X 131.26, Y 237.55, Z 0.00, A 0, B 0, C 0} C_DIS
LIN {X 131.26, Y 237.87, Z 0.00, A 0, B 0, C 0} C_DIS
LIN {X 131.26, Y 238.20, Z 0.00, A 0, B 0, C 0} C_DIS
LIN {X 131.26, Y 238.53, Z 0.00, A 0, B 0, C 0} C_DIS
LIN {X 131.26, Y 238.86, Z 0.00, A 0, B 0, C 0} C_DIS
LIN {X 131.26, Y 239.18, Z 0.00, A 0, B 0, C 0} C_DIS
LIN {X 131.26, Y 239.51, Z 0.00, A 0, B 0, C 0} C_DIS
LIN {X 131.26, Y 239.84, Z 0.00, A 0, B 0, C 0} C_DIS
LIN {X 131.26, Y 240.17, Z 0.00, A 0, B 0, C 0} C_DIS
LIN {X 131.26, Y 240.50, Z 0.00, A 0, B 0, C 0} C_DIS
LIN {X 131.26, Y 240.82, Z 0.00, A 0, B 0, C 0} C_DIS
LIN {X 131.26, Y 241.15, Z 0.00, A 0, B 0, C 0} C_DIS
LIN {X 131.26, Y 241.48, Z 0.00, A 0, B 0, C 0} C_DIS
LIN {X 131.26, Y 241.81, Z 0.00, A 0, B 0, C 0} C_DIS
LIN {X 131.26, Y 242.13, Z 0.00, A 0, B 0, C 0} C_DIS
LIN {X 131.26, Y 242.46, Z 0.00, A 0, B 0, C 0} C_DIS
LIN {X 131.26, Y 242.79, Z 0.00, A 0, B 0, C 0} C_DIS
LIN {X 131.26, Y 243.12, Z 0.00, A 0, B 0, C 0} C_DIS
LIN {X 131.26, Y 243.45, Z 0.00, A 0, B 0, C 0} C_DIS
LIN {X 131.26, Y 243.77, Z 0.00, A 0, B 0, C 0} C_DIS
LIN {X 131.26, Y 244.10, Z 0.00, A 0, B 0, C 0} C_DIS
LIN {X 131.26, Y 244.43, Z 0.00, A 0, B 0, C 0} C_DIS
LIN {X 131.26, Y 244.76, Z 0.00, A 0, B 0, C 0} C_DIS
LIN {X 131.26, Y 245.08, Z 0.00, A 0, B 0, C 0} C_DIS
LIN {X 131.26, Y 245.41, Z 0.00, A 0, B 0, C 0} C_DIS
LIN {X 131.26, Y 245.74, Z 0.00, A 0, B 0, C 0} C_DIS
LIN {X 131.26, Y 246.07, Z 0.00, A 0, B 0, C 0} C_DIS
LIN {X 131.26, Y 246.39, Z 0.00, A 0, B 0, C 0} C_DIS
LIN {X 131.26, Y 246.72, Z 0.00, A 0, B 0, C 0} C_DIS
LIN {X 131.26, Y 247.05, Z 0.00, A 0, B 0, C 0} C_DIS
LIN {X 131.26, Y 247.38, Z 0.00, A 0, B 0, C 0} C_DIS
LIN {X 131.26, Y 247.71, Z 0.00, A 0, B 0, C 0} C_DIS
LIN {X 131.26, Y 248.03, Z 0.00, A 0, B 0, C 0} C_DIS
LIN {X 131.26, Y 248.36, Z 0.00, A 0, B 0, C 0} C_DIS
LIN {X 131.26, Y 248.69, Z 0.00, A 0, B 0, C 0} C_DIS
LIN {X 131.26, Y 249.02, Z 0.00, A 0, B 0, C 0} C_DIS
LIN {X 131.26, Y 249.34, Z 0.00, A 0, B 0, C 0} C_DIS
LIN {X 131.26, Y 249.67, Z 0.00, A 0, B 0, C 0} C_DIS
LIN {X 131.26, Y 250.00, Z 0.00, A 0, B 0, C 0} C_DIS
LIN {X 131.26, Y 250.33, Z 0.00, A 0, B 0, C 0} C_DIS
LIN {X 131.26, Y 250.65, Z 0.00, A 0, B 0, C 0} C_DIS
LIN {X 131.26, Y 250.98, Z 0.00, A 0, B 0, C 0} C_DIS
LIN {X 131.26, Y 251.31, Z 0.00, A 0, B 0, C 0} C_DIS
LIN {X 131.26, Y 251.64, Z 0.00, A 0, B 0, C 0} C_DIS
LIN {X 131.26, Y 251.97, Z 0.00, A 0, B 0, C 0} C_DIS
LIN {X 131.26, Y 252.29, Z 0.00, A 0, B 0, C 0} C_DIS
LIN {X 131.26, Y 252.62, Z 0.00, A 0, B 0, C 0} C_DIS
LIN {X 131.26, Y 252.95, Z 0.00, A 0, B 0, C 0} C_DIS
LIN {X 131.26, Y 253.28, Z 0.00, A 0, B 0, C 0} C_DIS
LIN {X 131.26, Y 253.60, Z 0.00, A 0, B 0, C 0} C_DIS
LIN {X 131.26, Y 253.93, Z 0.00, A 0, B 0, C 0} C_DIS
LIN {X 131.27, Y 254.26, Z 0.00, A 0, B 0, C 0} C_DIS
LIN {X 131.29, Y 254.58, Z 0.00, A 0, B 0, C 0} C_DIS
LIN {X 131.32, Y 254.91, Z 0.00, A 0, B 0, C 0} C_DIS
LIN {X 131.37, Y 255.23, Z 0.00, A 0, B 0, C 0} C_DIS
LIN {X 131.43, Y 255.54, Z 0.00, A 0, B 0, C 0} C_DIS
LIN {X 131.49, Y 255.86, Z 0.00, A 0, B 0, C 0} C_DIS
LIN {X 131.57, Y 256.17, Z 0.00, A 0, B 0, C 0} C_DIS
LIN {X 131.68, Y 256.43, Z 0.00, A 0, B 0, C 0} C_DIS
LIN {X 131.84, Y 256.66, Z 0.00, A 0, B 0, C 0} C_DIS
LIN {X 132.00, Y 256.90, Z 0.00, A 0, B 0, C 0} C_DIS
LIN {X 132.15, Y 257.15, Z 0.00, A 0, B 0, C 0} C_DIS
LIN {X 132.31, Y 257.35, Z 0.00, A 0, B 0, C 0} C_DIS
LIN {X 132.51, Y 257.48, Z 0.00, A 0, B 0, C 0} C_DIS
LIN {X 132.71, Y 257.58, Z 0.00, A 0, B 0, C 0} C_DIS
LIN {X 132.92, Y 257.68, Z 0.00, A 0, B 0, C 0} C_DIS
LIN {X 133.14, Y 257.76, Z 0.00, A 0, B 0, C 0} C_DIS
LIN {X 133.35, Y 257.82, Z 0.00, A 0, B 0, C 0} C_DIS
LIN {X 133.56, Y 257.86, Z 0.00, A 0, B 0, C 0} C_DIS
LIN {X 133.78, Y 257.87, Z 0.00, A 0, B 0, C 0} C_DIS
LIN {X 134.00, Y 257.88, Z 0.00, A 0, B 0, C 0} C_DIS
LIN {X 134.22, Y 257.88, Z 0.00, A 0, B 0, C 0} C_DIS
LIN {X 134.43, Y 257.88, Z 0.00, A 0, B 0, C 0} C_DIS
LIN {X 134.65, Y 257.89, Z 0.00, A 0, B 0, C 0} C_DIS
LIN {X 134.87, Y 257.88, Z 0.00, A 0, B 0, C 0} C_DIS
LIN {X 135.09, Y 257.88, Z 0.00, A 0, B 0, C 0} C_DIS
LIN {X 135.30, Y 257.88, Z 0.00, A 0, B 0, C 0} C_DIS
LIN {X 135.52, Y 257.88, Z 0.00, A 0, B 0, C 0} C_DIS
LIN {X 135.74, Y 257.88, Z 0.00, A 0, B 0, C 0} C_DIS
LIN {X 135.96, Y 257.88, Z 0.00, A 0, B 0, C 0} C_DIS
LIN {X 136.17, Y 257.88, Z 0.00, A 0, B 0, C 0} C_DIS
LIN {X 136.39, Y 257.88, Z 0.00, A 0, B 0, C 0} C_DIS
LIN {X 136.61, Y 257.88, Z 0.00, A 0, B 0, C 0} C_DIS
LIN {X 136.82, Y 257.88, Z 0.00, A 0, B 0, C 0} C_DIS
LIN {X 137.04, Y 257.88, Z 0.00, A 0, B 0, C 0} C_DIS
LIN {X 137.26, Y 257.88, Z 0.00, A 0, B 0, C 0} C_DIS
LIN {X 137.48, Y 257.88, Z 0.00, A 0, B 0, C 0} C_DIS
LIN {X 137.69, Y 257.88, Z 0.00, A 0, B 0, C 0} C_DIS
LIN {X 137.91, Y 257.88, Z 0.00, A 0, B 0, C 0} C_DIS
LIN {X 138.13, Y 257.88, Z 0.00, A 0, B 0, C 0} C_DIS
LIN {X 138.35, Y 257.88, Z 0.00, A 0, B 0, C 0} C_DIS
LIN {X 138.56, Y 257.88, Z 0.00, A 0, B 0, C 0} C_DIS
LIN {X 138.78, Y 257.88, Z 0.00, A 0, B 0, C 0} C_DIS
LIN {X 139.00, Y 257.88, Z 0.00, A 0, B 0, C 0} C_DIS
LIN {X 139.22, Y 257.88, Z 0.00, A 0, B 0, C 0} C_DIS
LIN {X 139.43, Y 257.88, Z 0.00, A 0, B 0, C 0} C_DIS
LIN {X 139.65, Y 257.88, Z 0.00, A 0, B 0, C 0} C_DIS
LIN {X 139.87, Y 257.88, Z 0.00, A 0, B 0, C 0} C_DIS
LIN {X 140.09, Y 257.88, Z 0.00, A 0, B 0, C 0} C_DIS
LIN {X 140.30, Y 257.88, Z 0.00, A 0, B 0, C 0} C_DIS
LIN {X 140.52, Y 257.88, Z 0.00, A 0, B 0, C 0} C_DIS
LIN {X 140.74, Y 257.88, Z 0.00, A 0, B 0, C 0} C_DIS
LIN {X 140.96, Y 257.88, Z 0.00, A 0, B 0, C 0} C_DIS
LIN {X 141.17, Y 257.88, Z 0.00, A 0, B 0, C 0} C_DIS
LIN {X 141.39, Y 257.88, Z 0.00, A 0, B 0, C 0} C_DIS
LIN {X 141.61, Y 257.88, Z 0.00, A 0, B 0, C 0} C_DIS
LIN {X 141.83, Y 257.88, Z 0.00, A 0, B 0, C 0} C_DIS
LIN {X 142.04, Y 257.88, Z 0.00, A 0, B 0, C 0} C_DIS
LIN {X 142.26, Y 257.88, Z 0.00, A 0, B 0, C 0} C_DIS
LIN {X 142.48, Y 257.88, Z 0.00, A 0, B 0, C 0} C_DIS
LIN {X 142.70, Y 257.88, Z 0.00, A 0, B 0, C 0} C_DIS
LIN {X 142.91, Y 257.88, Z 0.00, A 0, B 0, C 0} C_DIS
LIN {X 143.13, Y 257.88, Z 0.00, A 0, B 0, C 0} C_DIS
LIN {X 143.35, Y 257.88, Z 0.00, A 0, B 0, C 0} C_DIS
LIN {X 143.57, Y 257.88, Z 0.00, A 0, B 0, C 0} C_DIS
LIN {X 143.78, Y 257.88, Z 0.00, A 0, B 0, C 0} C_DIS
LIN {X 144.00, Y 257.88, Z 0.00, A 0, B 0, C 0} C_DIS
LIN {X 144.22, Y 257.88, Z 0.00, A 0, B 0, C 0} C_DIS
LIN {X 144.44, Y 257.88, Z 0.00, A 0, B 0, C 0} C_DIS
LIN {X 144.65, Y 257.88, Z 0.00, A 0, B 0, C 0} C_DIS
LIN {X 144.87, Y 257.88, Z 0.00, A 0, B 0, C 0} C_DIS
LIN {X 145.09, Y 257.88, Z 0.00, A 0, B 0, C 0} C_DIS
LIN {X 145.31, Y 257.88, Z 0.00, A 0, B 0, C 0} C_DIS
LIN {X 145.52, Y 257.88, Z 0.00, A 0, B 0, C 0} C_DIS
LIN {X 145.74, Y 257.88, Z 0.00, A 0, B 0, C 0} C_DIS
LIN {X 145.96, Y 257.88, Z 0.00, A 0, B 0, C 0} C_DIS
LIN {X 146.18, Y 257.88, Z 0.00, A 0, B 0, C 0} C_DIS
LIN {X 146.39, Y 257.88, Z 0.00, A 0, B 0, C 0} C_DIS
LIN {X 146.61, Y 257.88, Z 0.00, A 0, B 0, C 0} C_DIS
LIN {X 146.83, Y 257.88, Z 0.00, A 0, B 0, C 0} C_DIS
LIN {X 147.05, Y 257.88, Z 0.00, A 0, B 0, C 0} C_DIS
LIN {X 147.26, Y 257.88, Z 0.00, A 0, B 0, C 0} C_DIS
LIN {X 147.48, Y 257.88, Z 0.00, A 0, B 0, C 0} C_DIS
LIN {X 147.70, Y 257.88, Z 0.00, A 0, B 0, C 0} C_DIS
LIN {X 147.92, Y 257.88, Z 0.00, A 0, B 0, C 0} C_DIS
LIN {X 148.13, Y 257.88, Z 0.00, A 0, B 0, C 0} C_DIS
LIN {X 148.35, Y 257.88, Z 0.00, A 0, B 0, C 0} C_DIS
LIN {X 148.57, Y 257.88, Z 0.00, A 0, B 0, C 0} C_DIS
LIN {X 148.78, Y 257.88, Z 0.00, A 0, B 0, C 0} C_DIS
LIN {X 149.00, Y 257.88, Z 0.00, A 0, B 0, C 0} C_DIS
LIN {X 149.22, Y 257.88, Z 0.00, A 0, B 0, C 0} C_DIS
LIN {X 149.44, Y 257.88, Z 0.00, A 0, B 0, C 0} C_DIS
LIN {X 149.65, Y 257.88, Z 0.00, A 0, B 0, C 0} C_DIS
LIN {X 149.87, Y 257.88, Z 0.00, A 0, B 0, C 0} C_DIS
LIN {X 150.09, Y 257.88, Z 0.00, A 0, B 0, C 0} C_DIS
LIN {X 150.31, Y 257.88, Z 0.00, A 0, B 0, C 0} C_DIS
LIN {X 150.52, Y 257.88, Z 0.00, A 0, B 0, C 0} C_DIS
LIN {X 150.74, Y 257.88, Z 0.00, A 0, B 0, C 0} C_DIS
LIN {X 150.96, Y 257.88, Z 0.00, A 0, B 0, C 0} C_DIS
LIN {X 151.18, Y 257.88, Z 0.00, A 0, B 0, C 0} C_DIS
LIN {X 151.39, Y 257.88, Z 0.00, A 0, B 0, C 0} C_DIS
LIN {X 151.61, Y 257.88, Z 0.00, A 0, B 0, C 0} C_DIS
LIN {X 151.83, Y 257.88, Z 0.00, A 0, B 0, C 0} C_DIS
LIN {X 152.05, Y 257.88, Z 0.00, A 0, B 0, C 0} C_DIS
LIN {X 152.26, Y 257.88, Z 0.00, A 0, B 0, C 0} C_DIS
LIN {X 152.48, Y 257.88, Z 0.00, A 0, B 0, C 0} C_DIS
LIN {X 152.70, Y 257.88, Z 0.00, A 0, B 0, C 0} C_DIS
LIN {X 152.92, Y 257.88, Z 0.00, A 0, B 0, C 0} C_DIS
LIN {X 153.13, Y 257.88, Z 0.00, A 0, B 0, C 0} C_DIS
LIN {X 153.35, Y 257.88, Z 0.00, A 0, B 0, C 0} C_DIS
LIN {X 153.57, Y 257.88, Z 0.00, A 0, B 0, C 0} C_DIS
LIN {X 153.79, Y 257.88, Z 0.00, A 0, B 0, C 0} C_DIS
LIN {X 154.00, Y 257.89, Z 0.00, A 0, B 0, C 0} C_DIS
LIN {X 154.22, Y 257.89, Z 0.00, A 0, B 0, C 0} C_DIS
LIN {X 154.44, Y 257.89, Z 0.00, A 0, B 0, C 0} C_DIS
LIN {X 154.66, Y 257.89, Z 0.00, A 0, B 0, C 0} C_DIS
LIN {X 154.87, Y 257.89, Z 0.00, A 0, B 0, C 0} C_DIS
LIN {X 155.09, Y 257.88, Z 0.00, A 0, B 0, C 0} C_DIS
LIN {X 155.31, Y 257.88, Z 0.00, A 0, B 0, C 0} C_DIS
LIN {X 155.53, Y 257.88, Z 0.00, A 0, B 0, C 0} C_DIS
LIN {X 155.74, Y 257.87, Z 0.00, A 0, B 0, C 0} C_DIS
LIN {X 155.96, Y 257.86, Z 0.00, A 0, B 0, C 0} C_DIS
LIN {X 156.18, Y 257.83, Z 0.00, A 0, B 0, C 0} C_DIS
LIN {X 156.39, Y 257.79, Z 0.00, A 0, B 0, C 0} C_DIS
LIN {X 156.61, Y 257.73, Z 0.00, A 0, B 0, C 0} C_DIS
LIN {X 156.82, Y 257.64, Z 0.00, A 0, B 0, C 0} C_DIS
LIN {X 156.82, Y 257.64, Z 10.00, A 0, B 0, C 0}

; ----- Contour 4 -----
PTP {X 107.58, Y 84.97, Z 10.00, A 0, B 0, C 0}
LIN {X 107.58, Y 84.97, Z 0.00, A 0, B 0, C 0}
LIN {X 107.80, Y 84.95, Z 0.00, A 0, B 0, C 0} C_DIS
LIN {X 108.02, Y 84.94, Z 0.00, A 0, B 0, C 0} C_DIS
LIN {X 108.23, Y 84.91, Z 0.00, A 0, B 0, C 0} C_DIS
LIN {X 108.45, Y 84.89, Z 0.00, A 0, B 0, C 0} C_DIS
LIN {X 108.67, Y 84.85, Z 0.00, A 0, B 0, C 0} C_DIS
LIN {X 108.88, Y 84.82, Z 0.00, A 0, B 0, C 0} C_DIS
LIN {X 109.09, Y 84.77, Z 0.00, A 0, B 0, C 0} C_DIS
LIN {X 109.31, Y 84.72, Z 0.00, A 0, B 0, C 0} C_DIS
LIN {X 109.52, Y 84.66, Z 0.00, A 0, B 0, C 0} C_DIS
LIN {X 109.73, Y 84.60, Z 0.00, A 0, B 0, C 0} C_DIS
LIN {X 109.94, Y 84.52, Z 0.00, A 0, B 0, C 0} C_DIS
LIN {X 110.15, Y 84.44, Z 0.00, A 0, B 0, C 0} C_DIS
LIN {X 110.36, Y 84.35, Z 0.00, A 0, B 0, C 0} C_DIS
LIN {X 110.57, Y 84.25, Z 0.00, A 0, B 0, C 0} C_DIS
LIN {X 110.77, Y 84.14, Z 0.00, A 0, B 0, C 0} C_DIS
LIN {X 110.98, Y 84.03, Z 0.00, A 0, B 0, C 0} C_DIS
LIN {X 111.18, Y 83.92, Z 0.00, A 0, B 0, C 0} C_DIS
LIN {X 111.39, Y 83.81, Z 0.00, A 0, B 0, C 0} C_DIS
LIN {X 111.59, Y 83.70, Z 0.00, A 0, B 0, C 0} C_DIS
LIN {X 111.79, Y 83.59, Z 0.00, A 0, B 0, C 0} C_DIS
LIN {X 112.00, Y 83.48, Z 0.00, A 0, B 0, C 0} C_DIS
LIN {X 112.20, Y 83.37, Z 0.00, A 0, B 0, C 0} C_DIS
LIN {X 112.41, Y 83.27, Z 0.00, A 0, B 0, C 0} C_DIS
LIN {X 112.61, Y 83.16, Z 0.00, A 0, B 0, C 0} C_DIS
LIN {X 112.81, Y 83.03, Z 0.00, A 0, B 0, C 0} C_DIS
LIN {X 113.00, Y 82.90, Z 0.00, A 0, B 0, C 0} C_DIS
LIN {X 113.19, Y 82.74, Z 0.00, A 0, B 0, C 0} C_DIS
LIN {X 113.37, Y 82.56, Z 0.00, A 0, B 0, C 0} C_DIS
LIN {X 113.55, Y 82.37, Z 0.00, A 0, B 0, C 0} C_DIS
LIN {X 113.73, Y 82.17, Z 0.00, A 0, B 0, C 0} C_DIS
LIN {X 113.91, Y 81.98, Z 0.00, A 0, B 0, C 0} C_DIS
LIN {X 114.09, Y 81.80, Z 0.00, A 0, B 0, C 0} C_DIS
LIN {X 114.27, Y 81.63, Z 0.00, A 0, B 0, C 0} C_DIS
LIN {X 114.46, Y 81.47, Z 0.00, A 0, B 0, C 0} C_DIS
LIN {X 114.65, Y 81.32, Z 0.00, A 0, B 0, C 0} C_DIS
LIN {X 114.85, Y 81.17, Z 0.00, A 0, B 0, C 0} C_DIS
LIN {X 115.04, Y 81.02, Z 0.00, A 0, B 0, C 0} C_DIS
LIN {X 115.23, Y 80.87, Z 0.00, A 0, B 0, C 0} C_DIS
LIN {X 115.42, Y 80.71, Z 0.00, A 0, B 0, C 0} C_DIS
LIN {X 115.60, Y 80.53, Z 0.00, A 0, B 0, C 0} C_DIS
LIN {X 115.77, Y 80.34, Z 0.00, A 0, B 0, C 0} C_DIS
LIN {X 115.94, Y 80.13, Z 0.00, A 0, B 0, C 0} C_DIS
LIN {X 116.10, Y 79.90, Z 0.00, A 0, B 0, C 0} C_DIS
LIN {X 116.25, Y 79.67, Z 0.00, A 0, B 0, C 0} C_DIS
LIN {X 116.41, Y 79.44, Z 0.00, A 0, B 0, C 0} C_DIS
LIN {X 116.56, Y 79.20, Z 0.00, A 0, B 0, C 0} C_DIS
LIN {X 116.71, Y 78.97, Z 0.00, A 0, B 0, C 0} C_DIS
LIN {X 116.87, Y 78.74, Z 0.00, A 0, B 0, C 0} C_DIS
LIN {X 117.02, Y 78.52, Z 0.00, A 0, B 0, C 0} C_DIS
LIN {X 117.18, Y 78.29, Z 0.00, A 0, B 0, C 0} C_DIS
LIN {X 117.33, Y 78.06, Z 0.00, A 0, B 0, C 0} C_DIS
LIN {X 117.49, Y 77.83, Z 0.00, A 0, B 0, C 0} C_DIS
LIN {X 117.64, Y 77.59, Z 0.00, A 0, B 0, C 0} C_DIS
LIN {X 117.79, Y 77.36, Z 0.00, A 0, B 0, C 0} C_DIS
LIN {X 117.94, Y 77.11, Z 0.00, A 0, B 0, C 0} C_DIS
LIN {X 118.08, Y 76.87, Z 0.00, A 0, B 0, C 0} C_DIS
LIN {X 118.23, Y 76.62, Z 0.00, A 0, B 0, C 0} C_DIS
LIN {X 118.37, Y 76.37, Z 0.00, A 0, B 0, C 0} C_DIS
LIN {X 118.50, Y 76.12, Z 0.00, A 0, B 0, C 0} C_DIS
LIN {X 118.63, Y 75.86, Z 0.00, A 0, B 0, C 0} C_DIS
LIN {X 118.76, Y 75.59, Z 0.00, A 0, B 0, C 0} C_DIS
LIN {X 118.88, Y 75.32, Z 0.00, A 0, B 0, C 0} C_DIS
LIN {X 119.00, Y 75.05, Z 0.00, A 0, B 0, C 0} C_DIS
LIN {X 119.12, Y 74.78, Z 0.00, A 0, B 0, C 0} C_DIS
LIN {X 119.23, Y 74.50, Z 0.00, A 0, B 0, C 0} C_DIS
LIN {X 119.34, Y 74.22, Z 0.00, A 0, B 0, C 0} C_DIS
LIN {X 119.45, Y 73.94, Z 0.00, A 0, B 0, C 0} C_DIS
LIN {X 119.56, Y 73.66, Z 0.00, A 0, B 0, C 0} C_DIS
LIN {X 119.66, Y 73.37, Z 0.00, A 0, B 0, C 0} C_DIS
LIN {X 119.77, Y 73.08, Z 0.00, A 0, B 0, C 0} C_DIS
LIN {X 119.87, Y 72.79, Z 0.00, A 0, B 0, C 0} C_DIS
LIN {X 119.97, Y 72.50, Z 0.00, A 0, B 0, C 0} C_DIS
LIN {X 120.07, Y 72.21, Z 0.00, A 0, B 0, C 0} C_DIS
LIN {X 120.17, Y 71.92, Z 0.00, A 0, B 0, C 0} C_DIS
LIN {X 120.27, Y 71.63, Z 0.00, A 0, B 0, C 0} C_DIS
LIN {X 120.36, Y 71.34, Z 0.00, A 0, B 0, C 0} C_DIS
LIN {X 120.46, Y 71.05, Z 0.00, A 0, B 0, C 0} C_DIS
LIN {X 120.56, Y 70.75, Z 0.00, A 0, B 0, C 0} C_DIS
LIN {X 120.66, Y 70.46, Z 0.00, A 0, B 0, C 0} C_DIS
LIN {X 120.76, Y 70.17, Z 0.00, A 0, B 0, C 0} C_DIS
LIN {X 120.85, Y 69.88, Z 0.00, A 0, B 0, C 0} C_DIS
LIN {X 120.94, Y 69.58, Z 0.00, A 0, B 0, C 0} C_DIS
LIN {X 121.03, Y 69.29, Z 0.00, A 0, B 0, C 0} C_DIS
LIN {X 121.12, Y 68.99, Z 0.00, A 0, B 0, C 0} C_DIS
LIN {X 121.20, Y 68.69, Z 0.00, A 0, B 0, C 0} C_DIS
LIN {X 121.28, Y 68.39, Z 0.00, A 0, B 0, C 0} C_DIS
LIN {X 121.35, Y 68.08, Z 0.00, A 0, B 0, C 0} C_DIS
LIN {X 121.42, Y 67.77, Z 0.00, A 0, B 0, C 0} C_DIS
LIN {X 121.48, Y 67.46, Z 0.00, A 0, B 0, C 0} C_DIS
LIN {X 121.54, Y 67.14, Z 0.00, A 0, B 0, C 0} C_DIS
LIN {X 121.59, Y 66.83, Z 0.00, A 0, B 0, C 0} C_DIS
LIN {X 121.63, Y 66.51, Z 0.00, A 0, B 0, C 0} C_DIS
LIN {X 121.68, Y 66.18, Z 0.00, A 0, B 0, C 0} C_DIS
LIN {X 121.71, Y 65.86, Z 0.00, A 0, B 0, C 0} C_DIS
LIN {X 121.74, Y 65.54, Z 0.00, A 0, B 0, C 0} C_DIS
LIN {X 121.77, Y 65.21, Z 0.00, A 0, B 0, C 0} C_DIS
LIN {X 121.79, Y 64.89, Z 0.00, A 0, B 0, C 0} C_DIS
LIN {X 121.81, Y 64.56, Z 0.00, A 0, B 0, C 0} C_DIS
LIN {X 121.83, Y 64.24, Z 0.00, A 0, B 0, C 0} C_DIS
LIN {X 121.84, Y 63.92, Z 0.00, A 0, B 0, C 0} C_DIS
LIN {X 121.86, Y 63.59, Z 0.00, A 0, B 0, C 0} C_DIS
LIN {X 121.88, Y 63.27, Z 0.00, A 0, B 0, C 0} C_DIS
LIN {X 121.91, Y 62.95, Z 0.00, A 0, B 0, C 0} C_DIS
LIN {X 121.95, Y 62.63, Z 0.00, A 0, B 0, C 0} C_DIS
LIN {X 121.99, Y 62.31, Z 0.00, A 0, B 0, C 0} C_DIS
LIN {X 122.04, Y 61.99, Z 0.00, A 0, B 0, C 0} C_DIS
LIN {X 122.08, Y 61.67, Z 0.00, A 0, B 0, C 0} C_DIS
LIN {X 122.12, Y 61.34, Z 0.00, A 0, B 0, C 0} C_DIS
LIN {X 122.16, Y 61.02, Z 0.00, A 0, B 0, C 0} C_DIS
LIN {X 122.18, Y 60.70, Z 0.00, A 0, B 0, C 0} C_DIS
LIN {X 122.20, Y 60.37, Z 0.00, A 0, B 0, C 0} C_DIS
LIN {X 122.22, Y 60.05, Z 0.00, A 0, B 0, C 0} C_DIS
LIN {X 122.23, Y 59.72, Z 0.00, A 0, B 0, C 0} C_DIS
LIN {X 122.24, Y 59.40, Z 0.00, A 0, B 0, C 0} C_DIS
LIN {X 122.24, Y 59.07, Z 0.00, A 0, B 0, C 0} C_DIS
LIN {X 122.24, Y 58.74, Z 0.00, A 0, B 0, C 0} C_DIS
LIN {X 122.24, Y 58.42, Z 0.00, A 0, B 0, C 0} C_DIS
LIN {X 122.24, Y 58.09, Z 0.00, A 0, B 0, C 0} C_DIS
LIN {X 122.24, Y 57.76, Z 0.00, A 0, B 0, C 0} C_DIS
LIN {X 122.23, Y 57.43, Z 0.00, A 0, B 0, C 0} C_DIS
LIN {X 122.23, Y 57.11, Z 0.00, A 0, B 0, C 0} C_DIS
LIN {X 122.23, Y 56.78, Z 0.00, A 0, B 0, C 0} C_DIS
LIN {X 122.23, Y 56.45, Z 0.00, A 0, B 0, C 0} C_DIS
LIN {X 122.22, Y 56.12, Z 0.00, A 0, B 0, C 0} C_DIS
LIN {X 122.22, Y 55.79, Z 0.00, A 0, B 0, C 0} C_DIS
LIN {X 122.22, Y 55.47, Z 0.00, A 0, B 0, C 0} C_DIS
LIN {X 122.22, Y 55.14, Z 0.00, A 0, B 0, C 0} C_DIS
LIN {X 122.22, Y 54.81, Z 0.00, A 0, B 0, C 0} C_DIS
LIN {X 122.22, Y 54.48, Z 0.00, A 0, B 0, C 0} C_DIS
LIN {X 122.21, Y 54.16, Z 0.00, A 0, B 0, C 0} C_DIS
LIN {X 122.21, Y 53.83, Z 0.00, A 0, B 0, C 0} C_DIS
LIN {X 122.21, Y 53.50, Z 0.00, A 0, B 0, C 0} C_DIS
LIN {X 122.21, Y 53.17, Z 0.00, A 0, B 0, C 0} C_DIS
LIN {X 122.21, Y 52.84, Z 0.00, A 0, B 0, C 0} C_DIS
LIN {X 122.21, Y 52.52, Z 0.00, A 0, B 0, C 0} C_DIS
LIN {X 122.21, Y 52.19, Z 0.00, A 0, B 0, C 0} C_DIS
LIN {X 122.21, Y 51.86, Z 0.00, A 0, B 0, C 0} C_DIS
LIN {X 122.21, Y 51.53, Z 0.00, A 0, B 0, C 0} C_DIS
LIN {X 122.21, Y 51.21, Z 0.00, A 0, B 0, C 0} C_DIS
LIN {X 122.21, Y 50.88, Z 0.00, A 0, B 0, C 0} C_DIS
LIN {X 122.21, Y 50.55, Z 0.00, A 0, B 0, C 0} C_DIS
LIN {X 122.21, Y 50.22, Z 0.00, A 0, B 0, C 0} C_DIS
LIN {X 122.21, Y 49.90, Z 0.00, A 0, B 0, C 0} C_DIS
LIN {X 122.21, Y 49.57, Z 0.00, A 0, B 0, C 0} C_DIS
LIN {X 122.21, Y 49.24, Z 0.00, A 0, B 0, C 0} C_DIS
LIN {X 122.21, Y 48.91, Z 0.00, A 0, B 0, C 0} C_DIS
LIN {X 122.21, Y 48.59, Z 0.00, A 0, B 0, C 0} C_DIS
LIN {X 122.21, Y 48.26, Z 0.00, A 0, B 0, C 0} C_DIS
LIN {X 122.21, Y 47.93, Z 0.00, A 0, B 0, C 0} C_DIS
LIN {X 122.21, Y 47.60, Z 0.00, A 0, B 0, C 0} C_DIS
LIN {X 122.21, Y 47.28, Z 0.00, A 0, B 0, C 0} C_DIS
LIN {X 122.21, Y 46.95, Z 0.00, A 0, B 0, C 0} C_DIS
LIN {X 122.21, Y 46.62, Z 0.00, A 0, B 0, C 0} C_DIS
LIN {X 122.21, Y 46.29, Z 0.00, A 0, B 0, C 0} C_DIS
LIN {X 122.21, Y 45.97, Z 0.00, A 0, B 0, C 0} C_DIS
LIN {X 122.21, Y 45.64, Z 0.00, A 0, B 0, C 0} C_DIS
LIN {X 122.21, Y 45.31, Z 0.00, A 0, B 0, C 0} C_DIS
LIN {X 122.21, Y 44.98, Z 0.00, A 0, B 0, C 0} C_DIS
LIN {X 122.21, Y 44.66, Z 0.00, A 0, B 0, C 0} C_DIS
LIN {X 122.21, Y 44.33, Z 0.00, A 0, B 0, C 0} C_DIS
LIN {X 122.21, Y 44.00, Z 0.00, A 0, B 0, C 0} C_DIS
LIN {X 122.21, Y 43.67, Z 0.00, A 0, B 0, C 0} C_DIS
LIN {X 122.21, Y 43.35, Z 0.00, A 0, B 0, C 0} C_DIS
LIN {X 122.22, Y 43.02, Z 0.00, A 0, B 0, C 0} C_DIS
LIN {X 122.22, Y 42.69, Z 0.00, A 0, B 0, C 0} C_DIS
LIN {X 122.22, Y 42.36, Z 0.00, A 0, B 0, C 0} C_DIS
LIN {X 122.22, Y 42.04, Z 0.00, A 0, B 0, C 0} C_DIS
LIN {X 122.22, Y 41.71, Z 0.00, A 0, B 0, C 0} C_DIS
LIN {X 122.22, Y 41.38, Z 0.00, A 0, B 0, C 0} C_DIS
LIN {X 122.22, Y 41.05, Z 0.00, A 0, B 0, C 0} C_DIS
LIN {X 122.22, Y 40.73, Z 0.00, A 0, B 0, C 0} C_DIS
LIN {X 122.22, Y 40.40, Z 0.00, A 0, B 0, C 0} C_DIS
LIN {X 122.22, Y 40.07, Z 0.00, A 0, B 0, C 0} C_DIS
LIN {X 122.22, Y 39.74, Z 0.00, A 0, B 0, C 0} C_DIS
LIN {X 122.22, Y 39.42, Z 0.00, A 0, B 0, C 0} C_DIS
LIN {X 122.22, Y 39.09, Z 0.00, A 0, B 0, C 0} C_DIS
LIN {X 122.22, Y 38.76, Z 0.00, A 0, B 0, C 0} C_DIS
LIN {X 122.22, Y 38.43, Z 0.00, A 0, B 0, C 0} C_DIS
LIN {X 122.22, Y 38.11, Z 0.00, A 0, B 0, C 0} C_DIS
LIN {X 122.22, Y 37.78, Z 0.00, A 0, B 0, C 0} C_DIS
LIN {X 122.22, Y 37.45, Z 0.00, A 0, B 0, C 0} C_DIS
LIN {X 122.22, Y 37.12, Z 0.00, A 0, B 0, C 0} C_DIS
LIN {X 122.22, Y 36.80, Z 0.00, A 0, B 0, C 0} C_DIS
LIN {X 122.22, Y 36.47, Z 0.00, A 0, B 0, C 0} C_DIS
LIN {X 122.22, Y 36.14, Z 0.00, A 0, B 0, C 0} C_DIS
LIN {X 122.22, Y 35.81, Z 0.00, A 0, B 0, C 0} C_DIS
LIN {X 122.22, Y 35.49, Z 0.00, A 0, B 0, C 0} C_DIS
LIN {X 122.22, Y 35.16, Z 0.00, A 0, B 0, C 0} C_DIS
LIN {X 122.22, Y 34.83, Z 0.00, A 0, B 0, C 0} C_DIS
LIN {X 122.22, Y 34.50, Z 0.00, A 0, B 0, C 0} C_DIS
LIN {X 122.22, Y 34.18, Z 0.00, A 0, B 0, C 0} C_DIS
LIN {X 122.22, Y 33.85, Z 0.00, A 0, B 0, C 0} C_DIS
LIN {X 122.22, Y 33.52, Z 0.00, A 0, B 0, C 0} C_DIS
LIN {X 122.22, Y 33.20, Z 0.00, A 0, B 0, C 0} C_DIS
LIN {X 122.22, Y 32.87, Z 0.00, A 0, B 0, C 0} C_DIS
LIN {X 122.22, Y 32.54, Z 0.00, A 0, B 0, C 0} C_DIS
LIN {X 122.22, Y 32.21, Z 0.00, A 0, B 0, C 0} C_DIS
LIN {X 122.22, Y 31.89, Z 0.00, A 0, B 0, C 0} C_DIS
LIN {X 122.22, Y 31.56, Z 0.00, A 0, B 0, C 0} C_DIS
LIN {X 122.22, Y 31.23, Z 0.00, A 0, B 0, C 0} C_DIS
LIN {X 122.22, Y 30.90, Z 0.00, A 0, B 0, C 0} C_DIS
LIN {X 122.22, Y 30.58, Z 0.00, A 0, B 0, C 0} C_DIS
LIN {X 122.22, Y 30.25, Z 0.00, A 0, B 0, C 0} C_DIS
LIN {X 122.22, Y 29.92, Z 0.00, A 0, B 0, C 0} C_DIS
LIN {X 122.21, Y 29.59, Z 0.00, A 0, B 0, C 0} C_DIS
LIN {X 122.21, Y 29.27, Z 0.00, A 0, B 0, C 0} C_DIS
LIN {X 122.21, Y 28.94, Z 0.00, A 0, B 0, C 0} C_DIS
LIN {X 122.21, Y 28.61, Z 0.00, A 0, B 0, C 0} C_DIS
LIN {X 122.21, Y 28.28, Z 0.00, A 0, B 0, C 0} C_DIS
LIN {X 122.21, Y 27.96, Z 0.00, A 0, B 0, C 0} C_DIS
LIN {X 122.21, Y 27.63, Z 0.00, A 0, B 0, C 0} C_DIS
LIN {X 122.21, Y 27.30, Z 0.00, A 0, B 0, C 0} C_DIS
LIN {X 122.21, Y 26.97, Z 0.00, A 0, B 0, C 0} C_DIS
LIN {X 122.21, Y 26.65, Z 0.00, A 0, B 0, C 0} C_DIS
LIN {X 122.21, Y 26.32, Z 0.00, A 0, B 0, C 0} C_DIS
LIN {X 122.21, Y 25.99, Z 0.00, A 0, B 0, C 0} C_DIS
LIN {X 122.21, Y 25.66, Z 0.00, A 0, B 0, C 0} C_DIS
LIN {X 122.21, Y 25.34, Z 0.00, A 0, B 0, C 0} C_DIS
LIN {X 122.21, Y 25.01, Z 0.00, A 0, B 0, C 0} C_DIS
LIN {X 122.21, Y 24.68, Z 0.00, A 0, B 0, C 0} C_DIS
LIN {X 122.21, Y 24.35, Z 0.00, A 0, B 0, C 0} C_DIS
LIN {X 122.21, Y 24.03, Z 0.00, A 0, B 0, C 0} C_DIS
LIN {X 122.21, Y 23.70, Z 0.00, A 0, B 0, C 0} C_DIS
LIN {X 122.21, Y 23.37, Z 0.00, A 0, B 0, C 0} C_DIS
LIN {X 122.21, Y 23.04, Z 0.00, A 0, B 0, C 0} C_DIS
LIN {X 122.21, Y 22.72, Z 0.00, A 0, B 0, C 0} C_DIS
LIN {X 122.21, Y 22.39, Z 0.00, A 0, B 0, C 0} C_DIS
LIN {X 122.21, Y 22.06, Z 0.00, A 0, B 0, C 0} C_DIS
LIN {X 122.21, Y 21.73, Z 0.00, A 0, B 0, C 0} C_DIS
LIN {X 122.21, Y 21.41, Z 0.00, A 0, B 0, C 0} C_DIS
LIN {X 122.21, Y 21.08, Z 0.00, A 0, B 0, C 0} C_DIS
LIN {X 122.21, Y 20.75, Z 0.00, A 0, B 0, C 0} C_DIS
LIN {X 122.21, Y 20.42, Z 0.00, A 0, B 0, C 0} C_DIS
LIN {X 122.21, Y 20.10, Z 0.00, A 0, B 0, C 0} C_DIS
LIN {X 122.21, Y 19.77, Z 0.00, A 0, B 0, C 0} C_DIS
LIN {X 122.21, Y 19.44, Z 0.00, A 0, B 0, C 0} C_DIS
LIN {X 122.21, Y 19.11, Z 0.00, A 0, B 0, C 0} C_DIS
LIN {X 122.21, Y 18.79, Z 0.00, A 0, B 0, C 0} C_DIS
LIN {X 122.21, Y 18.46, Z 0.00, A 0, B 0, C 0} C_DIS
LIN {X 122.21, Y 18.13, Z 0.00, A 0, B 0, C 0} C_DIS
LIN {X 122.21, Y 17.80, Z 0.00, A 0, B 0, C 0} C_DIS
LIN {X 122.21, Y 17.48, Z 0.00, A 0, B 0, C 0} C_DIS
LIN {X 122.21, Y 17.15, Z 0.00, A 0, B 0, C 0} C_DIS
LIN {X 122.21, Y 16.82, Z 0.00, A 0, B 0, C 0} C_DIS
LIN {X 122.21, Y 16.49, Z 0.00, A 0, B 0, C 0} C_DIS
LIN {X 122.21, Y 16.17, Z 0.00, A 0, B 0, C 0} C_DIS
LIN {X 122.21, Y 15.84, Z 0.00, A 0, B 0, C 0} C_DIS
LIN {X 122.21, Y 15.51, Z 0.00, A 0, B 0, C 0} C_DIS
LIN {X 122.21, Y 15.18, Z 0.00, A 0, B 0, C 0} C_DIS
LIN {X 122.21, Y 14.85, Z 0.00, A 0, B 0, C 0} C_DIS
LIN {X 122.21, Y 14.53, Z 0.00, A 0, B 0, C 0} C_DIS
LIN {X 122.21, Y 14.20, Z 0.00, A 0, B 0, C 0} C_DIS
LIN {X 122.21, Y 13.87, Z 0.00, A 0, B 0, C 0} C_DIS
LIN {X 122.22, Y 13.54, Z 0.00, A 0, B 0, C 0} C_DIS
LIN {X 122.22, Y 13.22, Z 0.00, A 0, B 0, C 0} C_DIS
LIN {X 122.22, Y 12.89, Z 0.00, A 0, B 0, C 0} C_DIS
LIN {X 122.22, Y 12.56, Z 0.00, A 0, B 0, C 0} C_DIS
LIN {X 122.22, Y 12.23, Z 0.00, A 0, B 0, C 0} C_DIS
LIN {X 122.22, Y 11.91, Z 0.00, A 0, B 0, C 0} C_DIS
LIN {X 122.22, Y 11.58, Z 0.00, A 0, B 0, C 0} C_DIS
LIN {X 122.22, Y 11.25, Z 0.00, A 0, B 0, C 0} C_DIS
LIN {X 122.22, Y 10.92, Z 0.00, A 0, B 0, C 0} C_DIS
LIN {X 122.23, Y 10.59, Z 0.00, A 0, B 0, C 0} C_DIS
LIN {X 122.23, Y 10.27, Z 0.00, A 0, B 0, C 0} C_DIS
LIN {X 122.23, Y 9.94, Z 0.00, A 0, B 0, C 0} C_DIS
LIN {X 122.23, Y 9.61, Z 0.00, A 0, B 0, C 0} C_DIS
LIN {X 122.23, Y 9.28, Z 0.00, A 0, B 0, C 0} C_DIS
LIN {X 122.23, Y 8.96, Z 0.00, A 0, B 0, C 0} C_DIS
LIN {X 122.23, Y 8.63, Z 0.00, A 0, B 0, C 0} C_DIS
LIN {X 122.24, Y 8.30, Z 0.00, A 0, B 0, C 0} C_DIS
LIN {X 122.24, Y 7.97, Z 0.00, A 0, B 0, C 0} C_DIS
LIN {X 122.24, Y 7.65, Z 0.00, A 0, B 0, C 0} C_DIS
LIN {X 122.24, Y 7.32, Z 0.00, A 0, B 0, C 0} C_DIS
LIN {X 122.24, Y 6.99, Z 0.00, A 0, B 0, C 0} C_DIS
LIN {X 122.23, Y 6.66, Z 0.00, A 0, B 0, C 0} C_DIS
LIN {X 122.23, Y 6.34, Z 0.00, A 0, B 0, C 0} C_DIS
LIN {X 122.22, Y 6.01, Z 0.00, A 0, B 0, C 0} C_DIS
LIN {X 122.20, Y 5.69, Z 0.00, A 0, B 0, C 0} C_DIS
LIN {X 122.18, Y 5.36, Z 0.00, A 0, B 0, C 0} C_DIS
LIN {X 122.16, Y 5.04, Z 0.00, A 0, B 0, C 0} C_DIS
LIN {X 122.13, Y 4.72, Z 0.00, A 0, B 0, C 0} C_DIS
LIN {X 122.10, Y 4.40, Z 0.00, A 0, B 0, C 0} C_DIS
LIN {X 122.06, Y 4.08, Z 0.00, A 0, B 0, C 0} C_DIS
LIN {X 122.01, Y 3.76, Z 0.00, A 0, B 0, C 0} C_DIS
LIN {X 121.95, Y 3.45, Z 0.00, A 0, B 0, C 0} C_DIS
LIN {X 121.88, Y 3.15, Z 0.00, A 0, B 0, C 0} C_DIS
LIN {X 121.78, Y 2.86, Z 0.00, A 0, B 0, C 0} C_DIS
LIN {X 121.65, Y 2.60, Z 0.00, A 0, B 0, C 0} C_DIS
LIN {X 121.49, Y 2.37, Z 0.00, A 0, B 0, C 0} C_DIS
LIN {X 121.31, Y 2.17, Z 0.00, A 0, B 0, C 0} C_DIS
LIN {X 121.12, Y 2.02, Z 0.00, A 0, B 0, C 0} C_DIS
LIN {X 120.91, Y 1.92, Z 0.00, A 0, B 0, C 0} C_DIS
LIN {X 120.70, Y 1.87, Z 0.00, A 0, B 0, C 0} C_DIS
LIN {X 120.48, Y 1.87, Z 0.00, A 0, B 0, C 0} C_DIS
LIN {X 120.27, Y 1.91, Z 0.00, A 0, B 0, C 0} C_DIS
LIN {X 120.06, Y 1.98, Z 0.00, A 0, B 0, C 0} C_DIS
LIN {X 119.86, Y 2.08, Z 0.00, A 0, B 0, C 0} C_DIS
LIN {X 119.65, Y 2.18, Z 0.00, A 0, B 0, C 0} C_DIS
LIN {X 119.45, Y 2.30, Z 0.00, A 0, B 0, C 0} C_DIS
LIN {X 119.24, Y 2.41, Z 0.00, A 0, B 0, C 0} C_DIS
LIN {X 119.04, Y 2.52, Z 0.00, A 0, B 0, C 0} C_DIS
LIN {X 118.83, Y 2.62, Z 0.00, A 0, B 0, C 0} C_DIS
LIN {X 118.62, Y 2.71, Z 0.00, A 0, B 0, C 0} C_DIS
LIN {X 118.42, Y 2.81, Z 0.00, A 0, B 0, C 0} C_DIS
LIN {X 118.21, Y 2.91, Z 0.00, A 0, B 0, C 0} C_DIS
LIN {X 118.01, Y 3.03, Z 0.00, A 0, B 0, C 0} C_DIS
LIN {X 117.81, Y 3.15, Z 0.00, A 0, B 0, C 0} C_DIS
LIN {X 117.61, Y 3.29, Z 0.00, A 0, B 0, C 0} C_DIS
LIN {X 117.42, Y 3.43, Z 0.00, A 0, B 0, C 0} C_DIS
LIN {X 117.23, Y 3.59, Z 0.00, A 0, B 0, C 0} C_DIS
LIN {X 117.05, Y 3.76, Z 0.00, A 0, B 0, C 0} C_DIS
LIN {X 116.86, Y 3.94, Z 0.00, A 0, B 0, C 0} C_DIS
LIN {X 116.68, Y 4.13, Z 0.00, A 0, B 0, C 0} C_DIS
LIN {X 116.51, Y 4.32, Z 0.00, A 0, B 0, C 0} C_DIS
LIN {X 116.33, Y 4.51, Z 0.00, A 0, B 0, C 0} C_DIS
LIN {X 116.15, Y 4.70, Z 0.00, A 0, B 0, C 0} C_DIS
LIN {X 115.97, Y 4.88, Z 0.00, A 0, B 0, C 0} C_DIS
LIN {X 115.79, Y 5.07, Z 0.00, A 0, B 0, C 0} C_DIS
LIN {X 115.61, Y 5.25, Z 0.00, A 0, B 0, C 0} C_DIS
LIN {X 115.43, Y 5.42, Z 0.00, A 0, B 0, C 0} C_DIS
LIN {X 115.24, Y 5.59, Z 0.00, A 0, B 0, C 0} C_DIS
LIN {X 115.05, Y 5.76, Z 0.00, A 0, B 0, C 0} C_DIS
LIN {X 114.87, Y 5.93, Z 0.00, A 0, B 0, C 0} C_DIS
LIN {X 114.68, Y 6.11, Z 0.00, A 0, B 0, C 0} C_DIS
LIN {X 114.51, Y 6.30, Z 0.00, A 0, B 0, C 0} C_DIS
LIN {X 114.34, Y 6.50, Z 0.00, A 0, B 0, C 0} C_DIS
LIN {X 114.18, Y 6.72, Z 0.00, A 0, B 0, C 0} C_DIS
LIN {X 114.02, Y 6.94, Z 0.00, A 0, B 0, C 0} C_DIS
LIN {X 113.86, Y 7.16, Z 0.00, A 0, B 0, C 0} C_DIS
LIN {X 113.70, Y 7.38, Z 0.00, A 0, B 0, C 0} C_DIS
LIN {X 113.54, Y 7.61, Z 0.00, A 0, B 0, C 0} C_DIS
LIN {X 113.39, Y 7.84, Z 0.00, A 0, B 0, C 0} C_DIS
LIN {X 113.23, Y 8.06, Z 0.00, A 0, B 0, C 0} C_DIS
LIN {X 113.08, Y 8.29, Z 0.00, A 0, B 0, C 0} C_DIS
LIN {X 112.92, Y 8.52, Z 0.00, A 0, B 0, C 0} C_DIS
LIN {X 112.77, Y 8.75, Z 0.00, A 0, B 0, C 0} C_DIS
LIN {X 112.61, Y 8.98, Z 0.00, A 0, B 0, C 0} C_DIS
LIN {X 112.46, Y 9.21, Z 0.00, A 0, B 0, C 0} C_DIS
LIN {X 112.30, Y 9.44, Z 0.00, A 0, B 0, C 0} C_DIS
LIN {X 112.15, Y 9.67, Z 0.00, A 0, B 0, C 0} C_DIS
LIN {X 112.00, Y 9.90, Z 0.00, A 0, B 0, C 0} C_DIS
LIN {X 111.84, Y 10.14, Z 0.00, A 0, B 0, C 0} C_DIS
LIN {X 111.69, Y 10.37, Z 0.00, A 0, B 0, C 0} C_DIS
LIN {X 111.54, Y 10.60, Z 0.00, A 0, B 0, C 0} C_DIS
LIN {X 111.38, Y 10.83, Z 0.00, A 0, B 0, C 0} C_DIS
LIN {X 111.23, Y 11.07, Z 0.00, A 0, B 0, C 0} C_DIS
LIN {X 111.08, Y 11.30, Z 0.00, A 0, B 0, C 0} C_DIS
LIN {X 110.92, Y 11.53, Z 0.00, A 0, B 0, C 0} C_DIS
LIN {X 110.77, Y 11.76, Z 0.00, A 0, B 0, C 0} C_DIS
LIN {X 110.62, Y 11.99, Z 0.00, A 0, B 0, C 0} C_DIS
LIN {X 110.46, Y 12.23, Z 0.00, A 0, B 0, C 0} C_DIS
LIN {X 110.31, Y 12.46, Z 0.00, A 0, B 0, C 0} C_DIS
LIN {X 110.16, Y 12.69, Z 0.00, A 0, B 0, C 0} C_DIS
LIN {X 110.00, Y 12.92, Z 0.00, A 0, B 0, C 0} C_DIS
LIN {X 109.85, Y 13.16, Z 0.00, A 0, B 0, C 0} C_DIS
LIN {X 109.70, Y 13.39, Z 0.00, A 0, B 0, C 0} C_DIS
LIN {X 109.54, Y 13.62, Z 0.00, A 0, B 0, C 0} C_DIS
LIN {X 109.39, Y 13.85, Z 0.00, A 0, B 0, C 0} C_DIS
LIN {X 109.24, Y 14.08, Z 0.00, A 0, B 0, C 0} C_DIS
LIN {X 109.08, Y 14.31, Z 0.00, A 0, B 0, C 0} C_DIS
LIN {X 108.93, Y 14.55, Z 0.00, A 0, B 0, C 0} C_DIS
LIN {X 108.77, Y 14.78, Z 0.00, A 0, B 0, C 0} C_DIS
LIN {X 108.62, Y 15.01, Z 0.00, A 0, B 0, C 0} C_DIS
LIN {X 108.47, Y 15.24, Z 0.00, A 0, B 0, C 0} C_DIS
LIN {X 108.31, Y 15.47, Z 0.00, A 0, B 0, C 0} C_DIS
LIN {X 108.16, Y 15.71, Z 0.00, A 0, B 0, C 0} C_DIS
LIN {X 108.01, Y 15.94, Z 0.00, A 0, B 0, C 0} C_DIS
LIN {X 107.85, Y 16.17, Z 0.00, A 0, B 0, C 0} C_DIS
LIN {X 107.70, Y 16.40, Z 0.00, A 0, B 0, C 0} C_DIS
LIN {X 107.55, Y 16.63, Z 0.00, A 0, B 0, C 0} C_DIS
LIN {X 107.39, Y 16.86, Z 0.00, A 0, B 0, C 0} C_DIS
LIN {X 107.24, Y 17.09, Z 0.00, A 0, B 0, C 0} C_DIS
LIN {X 107.08, Y 17.33, Z 0.00, A 0, B 0, C 0} C_DIS
LIN {X 106.93, Y 17.56, Z 0.00, A 0, B 0, C 0} C_DIS
LIN {X 106.78, Y 17.79, Z 0.00, A 0, B 0, C 0} C_DIS
LIN {X 106.62, Y 18.02, Z 0.00, A 0, B 0, C 0} C_DIS
LIN {X 106.47, Y 18.25, Z 0.00, A 0, B 0, C 0} C_DIS
LIN {X 106.32, Y 18.48, Z 0.00, A 0, B 0, C 0} C_DIS
LIN {X 106.16, Y 18.72, Z 0.00, A 0, B 0, C 0} C_DIS
LIN {X 106.01, Y 18.95, Z 0.00, A 0, B 0, C 0} C_DIS
LIN {X 105.85, Y 19.18, Z 0.00, A 0, B 0, C 0} C_DIS
LIN {X 105.70, Y 19.41, Z 0.00, A 0, B 0, C 0} C_DIS
LIN {X 105.55, Y 19.64, Z 0.00, A 0, B 0, C 0} C_DIS
LIN {X 105.39, Y 19.87, Z 0.00, A 0, B 0, C 0} C_DIS
LIN {X 105.24, Y 20.10, Z 0.00, A 0, B 0, C 0} C_DIS
LIN {X 105.09, Y 20.34, Z 0.00, A 0, B 0, C 0} C_DIS
LIN {X 104.93, Y 20.57, Z 0.00, A 0, B 0, C 0} C_DIS
LIN {X 104.78, Y 20.80, Z 0.00, A 0, B 0, C 0} C_DIS
LIN {X 104.62, Y 21.03, Z 0.00, A 0, B 0, C 0} C_DIS
LIN {X 104.47, Y 21.26, Z 0.00, A 0, B 0, C 0} C_DIS
LIN {X 104.32, Y 21.49, Z 0.00, A 0, B 0, C 0} C_DIS
LIN {X 104.16, Y 21.72, Z 0.00, A 0, B 0, C 0} C_DIS
LIN {X 104.01, Y 21.95, Z 0.00, A 0, B 0, C 0} C_DIS
LIN {X 103.86, Y 22.19, Z 0.00, A 0, B 0, C 0} C_DIS
LIN {X 103.70, Y 22.42, Z 0.00, A 0, B 0, C 0} C_DIS
LIN {X 103.55, Y 22.65, Z 0.00, A 0, B 0, C 0} C_DIS
LIN {X 103.39, Y 22.88, Z 0.00, A 0, B 0, C 0} C_DIS
LIN {X 103.24, Y 23.11, Z 0.00, A 0, B 0, C 0} C_DIS
LIN {X 103.09, Y 23.34, Z 0.00, A 0, B 0, C 0} C_DIS
LIN {X 102.93, Y 23.57, Z 0.00, A 0, B 0, C 0} C_DIS
LIN {X 102.78, Y 23.81, Z 0.00, A 0, B 0, C 0} C_DIS
LIN {X 102.63, Y 24.04, Z 0.00, A 0, B 0, C 0} C_DIS
LIN {X 102.47, Y 24.27, Z 0.00, A 0, B 0, C 0} C_DIS
LIN {X 102.32, Y 24.50, Z 0.00, A 0, B 0, C 0} C_DIS
LIN {X 102.16, Y 24.73, Z 0.00, A 0, B 0, C 0} C_DIS
LIN {X 102.01, Y 24.96, Z 0.00, A 0, B 0, C 0} C_DIS
LIN {X 101.86, Y 25.19, Z 0.00, A 0, B 0, C 0} C_DIS
LIN {X 101.70, Y 25.43, Z 0.00, A 0, B 0, C 0} C_DIS
LIN {X 101.55, Y 25.66, Z 0.00, A 0, B 0, C 0} C_DIS
LIN {X 101.40, Y 25.89, Z 0.00, A 0, B 0, C 0} C_DIS
LIN {X 101.24, Y 26.12, Z 0.00, A 0, B 0, C 0} C_DIS
LIN {X 101.09, Y 26.35, Z 0.00, A 0, B 0, C 0} C_DIS
LIN {X 100.94, Y 26.58, Z 0.00, A 0, B 0, C 0} C_DIS
LIN {X 100.78, Y 26.82, Z 0.00, A 0, B 0, C 0} C_DIS
LIN {X 100.63, Y 27.05, Z 0.00, A 0, B 0, C 0} C_DIS
LIN {X 100.48, Y 27.28, Z 0.00, A 0, B 0, C 0} C_DIS
LIN {X 100.32, Y 27.51, Z 0.00, A 0, B 0, C 0} C_DIS
LIN {X 100.17, Y 27.74, Z 0.00, A 0, B 0, C 0} C_DIS
LIN {X 100.01, Y 27.97, Z 0.00, A 0, B 0, C 0} C_DIS
LIN {X 99.86, Y 28.21, Z 0.00, A 0, B 0, C 0} C_DIS
LIN {X 99.71, Y 28.44, Z 0.00, A 0, B 0, C 0} C_DIS
LIN {X 99.55, Y 28.67, Z 0.00, A 0, B 0, C 0} C_DIS
LIN {X 99.40, Y 28.90, Z 0.00, A 0, B 0, C 0} C_DIS
LIN {X 99.25, Y 29.13, Z 0.00, A 0, B 0, C 0} C_DIS
LIN {X 99.09, Y 29.37, Z 0.00, A 0, B 0, C 0} C_DIS
LIN {X 98.94, Y 29.60, Z 0.00, A 0, B 0, C 0} C_DIS
LIN {X 98.79, Y 29.83, Z 0.00, A 0, B 0, C 0} C_DIS
LIN {X 98.63, Y 30.06, Z 0.00, A 0, B 0, C 0} C_DIS
LIN {X 98.48, Y 30.29, Z 0.00, A 0, B 0, C 0} C_DIS
LIN {X 98.33, Y 30.53, Z 0.00, A 0, B 0, C 0} C_DIS
LIN {X 98.17, Y 30.76, Z 0.00, A 0, B 0, C 0} C_DIS
LIN {X 98.02, Y 30.99, Z 0.00, A 0, B 0, C 0} C_DIS
LIN {X 97.87, Y 31.22, Z 0.00, A 0, B 0, C 0} C_DIS
LIN {X 97.71, Y 31.45, Z 0.00, A 0, B 0, C 0} C_DIS
LIN {X 97.56, Y 31.68, Z 0.00, A 0, B 0, C 0} C_DIS
LIN {X 97.41, Y 31.92, Z 0.00, A 0, B 0, C 0} C_DIS
LIN {X 97.25, Y 32.15, Z 0.00, A 0, B 0, C 0} C_DIS
LIN {X 97.10, Y 32.38, Z 0.00, A 0, B 0, C 0} C_DIS
LIN {X 96.94, Y 32.61, Z 0.00, A 0, B 0, C 0} C_DIS
LIN {X 96.79, Y 32.84, Z 0.00, A 0, B 0, C 0} C_DIS
LIN {X 96.64, Y 33.07, Z 0.00, A 0, B 0, C 0} C_DIS
LIN {X 96.48, Y 33.30, Z 0.00, A 0, B 0, C 0} C_DIS
LIN {X 96.33, Y 33.54, Z 0.00, A 0, B 0, C 0} C_DIS
LIN {X 96.17, Y 33.77, Z 0.00, A 0, B 0, C 0} C_DIS
LIN {X 96.02, Y 34.00, Z 0.00, A 0, B 0, C 0} C_DIS
LIN {X 95.87, Y 34.23, Z 0.00, A 0, B 0, C 0} C_DIS
LIN {X 95.71, Y 34.46, Z 0.00, A 0, B 0, C 0} C_DIS
LIN {X 95.56, Y 34.69, Z 0.00, A 0, B 0, C 0} C_DIS
LIN {X 95.40, Y 34.92, Z 0.00, A 0, B 0, C 0} C_DIS
LIN {X 95.25, Y 35.15, Z 0.00, A 0, B 0, C 0} C_DIS
LIN {X 95.09, Y 35.38, Z 0.00, A 0, B 0, C 0} C_DIS
LIN {X 94.94, Y 35.61, Z 0.00, A 0, B 0, C 0} C_DIS
LIN {X 94.78, Y 35.84, Z 0.00, A 0, B 0, C 0} C_DIS
LIN {X 94.63, Y 36.07, Z 0.00, A 0, B 0, C 0} C_DIS
LIN {X 94.48, Y 36.30, Z 0.00, A 0, B 0, C 0} C_DIS
LIN {X 94.32, Y 36.53, Z 0.00, A 0, B 0, C 0} C_DIS
LIN {X 94.17, Y 36.77, Z 0.00, A 0, B 0, C 0} C_DIS
LIN {X 94.02, Y 37.00, Z 0.00, A 0, B 0, C 0} C_DIS
LIN {X 93.87, Y 37.24, Z 0.00, A 0, B 0, C 0} C_DIS
LIN {X 93.72, Y 37.48, Z 0.00, A 0, B 0, C 0} C_DIS
LIN {X 93.58, Y 37.72, Z 0.00, A 0, B 0, C 0} C_DIS
LIN {X 93.44, Y 37.97, Z 0.00, A 0, B 0, C 0} C_DIS
LIN {X 93.30, Y 38.23, Z 0.00, A 0, B 0, C 0} C_DIS
LIN {X 93.17, Y 38.48, Z 0.00, A 0, B 0, C 0} C_DIS
LIN {X 93.04, Y 38.75, Z 0.00, A 0, B 0, C 0} C_DIS
LIN {X 92.92, Y 39.02, Z 0.00, A 0, B 0, C 0} C_DIS
LIN {X 92.80, Y 39.29, Z 0.00, A 0, B 0, C 0} C_DIS
LIN {X 92.68, Y 39.56, Z 0.00, A 0, B 0, C 0} C_DIS
LIN {X 92.57, Y 39.84, Z 0.00, A 0, B 0, C 0} C_DIS
LIN {X 92.45, Y 40.12, Z 0.00, A 0, B 0, C 0} C_DIS
LIN {X 92.34, Y 40.40, Z 0.00, A 0, B 0, C 0} C_DIS
LIN {X 92.23, Y 40.68, Z 0.00, A 0, B 0, C 0} C_DIS
LIN {X 92.12, Y 40.96, Z 0.00, A 0, B 0, C 0} C_DIS
LIN {X 92.01, Y 41.25, Z 0.00, A 0, B 0, C 0} C_DIS
LIN {X 91.90, Y 41.53, Z 0.00, A 0, B 0, C 0} C_DIS
LIN {X 91.79, Y 41.82, Z 0.00, A 0, B 0, C 0} C_DIS
LIN {X 91.69, Y 42.10, Z 0.00, A 0, B 0, C 0} C_DIS
LIN {X 91.59, Y 42.39, Z 0.00, A 0, B 0, C 0} C_DIS
LIN {X 91.49, Y 42.68, Z 0.00, A 0, B 0, C 0} C_DIS
LIN {X 91.40, Y 42.98, Z 0.00, A 0, B 0, C 0} C_DIS
LIN {X 91.31, Y 43.27, Z 0.00, A 0, B 0, C 0} C_DIS
LIN {X 91.23, Y 43.57, Z 0.00, A 0, B 0, C 0} C_DIS
LIN {X 91.15, Y 43.87, Z 0.00, A 0, B 0, C 0} C_DIS
LIN {X 91.08, Y 44.18, Z 0.00, A 0, B 0, C 0} C_DIS
LIN {X 91.01, Y 44.49, Z 0.00, A 0, B 0, C 0} C_DIS
LIN {X 90.94, Y 44.80, Z 0.00, A 0, B 0, C 0} C_DIS
LIN {X 90.88, Y 45.11, Z 0.00, A 0, B 0, C 0} C_DIS
LIN {X 90.82, Y 45.42, Z 0.00, A 0, B 0, C 0} C_DIS
LIN {X 90.76, Y 45.74, Z 0.00, A 0, B 0, C 0} C_DIS
LIN {X 90.70, Y 46.06, Z 0.00, A 0, B 0, C 0} C_DIS
LIN {X 90.65, Y 46.37, Z 0.00, A 0, B 0, C 0} C_DIS
LIN {X 90.60, Y 46.69, Z 0.00, A 0, B 0, C 0} C_DIS
LIN {X 90.55, Y 47.01, Z 0.00, A 0, B 0, C 0} C_DIS
LIN {X 90.50, Y 47.33, Z 0.00, A 0, B 0, C 0} C_DIS
LIN {X 90.46, Y 47.66, Z 0.00, A 0, B 0, C 0} C_DIS
LIN {X 90.43, Y 47.98, Z 0.00, A 0, B 0, C 0} C_DIS
LIN {X 90.40, Y 48.30, Z 0.00, A 0, B 0, C 0} C_DIS
LIN {X 90.38, Y 48.63, Z 0.00, A 0, B 0, C 0} C_DIS
LIN {X 90.37, Y 48.95, Z 0.00, A 0, B 0, C 0} C_DIS
LIN {X 90.37, Y 49.28, Z 0.00, A 0, B 0, C 0} C_DIS
LIN {X 90.37, Y 49.61, Z 0.00, A 0, B 0, C 0} C_DIS
LIN {X 90.37, Y 49.93, Z 0.00, A 0, B 0, C 0} C_DIS
LIN {X 90.37, Y 50.26, Z 0.00, A 0, B 0, C 0} C_DIS
LIN {X 90.38, Y 50.59, Z 0.00, A 0, B 0, C 0} C_DIS
LIN {X 90.38, Y 50.92, Z 0.00, A 0, B 0, C 0} C_DIS
LIN {X 90.38, Y 51.24, Z 0.00, A 0, B 0, C 0} C_DIS
LIN {X 90.38, Y 51.57, Z 0.00, A 0, B 0, C 0} C_DIS
LIN {X 90.38, Y 51.90, Z 0.00, A 0, B 0, C 0} C_DIS
LIN {X 90.38, Y 52.23, Z 0.00, A 0, B 0, C 0} C_DIS
LIN {X 90.38, Y 52.56, Z 0.00, A 0, B 0, C 0} C_DIS
LIN {X 90.38, Y 52.88, Z 0.00, A 0, B 0, C 0} C_DIS
LIN {X 90.38, Y 53.21, Z 0.00, A 0, B 0, C 0} C_DIS
LIN {X 90.38, Y 53.54, Z 0.00, A 0, B 0, C 0} C_DIS
LIN {X 90.38, Y 53.87, Z 0.00, A 0, B 0, C 0} C_DIS
LIN {X 90.38, Y 54.19, Z 0.00, A 0, B 0, C 0} C_DIS
LIN {X 90.38, Y 54.52, Z 0.00, A 0, B 0, C 0} C_DIS
LIN {X 90.38, Y 54.85, Z 0.00, A 0, B 0, C 0} C_DIS
LIN {X 90.38, Y 55.18, Z 0.00, A 0, B 0, C 0} C_DIS
LIN {X 90.38, Y 55.50, Z 0.00, A 0, B 0, C 0} C_DIS
LIN {X 90.38, Y 55.83, Z 0.00, A 0, B 0, C 0} C_DIS
LIN {X 90.38, Y 56.16, Z 0.00, A 0, B 0, C 0} C_DIS
LIN {X 90.38, Y 56.48, Z 0.00, A 0, B 0, C 0} C_DIS
LIN {X 90.38, Y 56.81, Z 0.00, A 0, B 0, C 0} C_DIS
LIN {X 90.38, Y 57.14, Z 0.00, A 0, B 0, C 0} C_DIS
LIN {X 90.38, Y 57.47, Z 0.00, A 0, B 0, C 0} C_DIS
LIN {X 90.38, Y 57.79, Z 0.00, A 0, B 0, C 0} C_DIS
LIN {X 90.38, Y 58.12, Z 0.00, A 0, B 0, C 0} C_DIS
LIN {X 90.38, Y 58.45, Z 0.00, A 0, B 0, C 0} C_DIS
LIN {X 90.38, Y 58.78, Z 0.00, A 0, B 0, C 0} C_DIS
LIN {X 90.38, Y 59.10, Z 0.00, A 0, B 0, C 0} C_DIS
LIN {X 90.38, Y 59.43, Z 0.00, A 0, B 0, C 0} C_DIS
LIN {X 90.38, Y 59.76, Z 0.00, A 0, B 0, C 0} C_DIS
LIN {X 90.38, Y 60.09, Z 0.00, A 0, B 0, C 0} C_DIS
LIN {X 90.38, Y 60.41, Z 0.00, A 0, B 0, C 0} C_DIS
LIN {X 90.38, Y 60.74, Z 0.00, A 0, B 0, C 0} C_DIS
LIN {X 90.38, Y 61.07, Z 0.00, A 0, B 0, C 0} C_DIS
LIN {X 90.38, Y 61.40, Z 0.00, A 0, B 0, C 0} C_DIS
LIN {X 90.38, Y 61.73, Z 0.00, A 0, B 0, C 0} C_DIS
LIN {X 90.38, Y 62.05, Z 0.00, A 0, B 0, C 0} C_DIS
LIN {X 90.38, Y 62.38, Z 0.00, A 0, B 0, C 0} C_DIS
LIN {X 90.38, Y 62.71, Z 0.00, A 0, B 0, C 0} C_DIS
LIN {X 90.38, Y 63.04, Z 0.00, A 0, B 0, C 0} C_DIS
LIN {X 90.39, Y 63.36, Z 0.00, A 0, B 0, C 0} C_DIS
LIN {X 90.40, Y 63.69, Z 0.00, A 0, B 0, C 0} C_DIS
LIN {X 90.43, Y 64.01, Z 0.00, A 0, B 0, C 0} C_DIS
LIN {X 90.46, Y 64.33, Z 0.00, A 0, B 0, C 0} C_DIS
LIN {X 90.51, Y 64.65, Z 0.00, A 0, B 0, C 0} C_DIS
LIN {X 90.56, Y 64.97, Z 0.00, A 0, B 0, C 0} C_DIS
LIN {X 90.63, Y 65.28, Z 0.00, A 0, B 0, C 0} C_DIS
LIN {X 90.70, Y 65.59, Z 0.00, A 0, B 0, C 0} C_DIS
LIN {X 90.78, Y 65.90, Z 0.00, A 0, B 0, C 0} C_DIS
LIN {X 90.85, Y 66.21, Z 0.00, A 0, B 0, C 0} C_DIS
LIN {X 90.92, Y 66.52, Z 0.00, A 0, B 0, C 0} C_DIS
LIN {X 90.99, Y 66.83, Z 0.00, A 0, B 0, C 0} C_DIS
LIN {X 91.05, Y 67.14, Z 0.00, A 0, B 0, C 0} C_DIS
LIN {X 91.10, Y 67.46, Z 0.00, A 0, B 0, C 0} C_DIS
LIN {X 91.16, Y 67.77, Z 0.00, A 0, B 0, C 0} C_DIS
LIN {X 91.21, Y 68.09, Z 0.00, A 0, B 0, C 0} C_DIS
LIN {X 91.25, Y 68.41, Z 0.00, A 0, B 0, C 0} C_DIS
LIN {X 91.30, Y 68.73, Z 0.00, A 0, B 0, C 0} C_DIS
LIN {X 91.36, Y 69.05, Z 0.00, A 0, B 0, C 0} C_DIS
LIN {X 91.42, Y 69.36, Z 0.00, A 0, B 0, C 0} C_DIS
LIN {X 91.49, Y 69.67, Z 0.00, A 0, B 0, C 0} C_DIS
LIN {X 91.57, Y 69.97, Z 0.00, A 0, B 0, C 0} C_DIS
LIN {X 91.65, Y 70.27, Z 0.00, A 0, B 0, C 0} C_DIS
LIN {X 91.74, Y 70.57, Z 0.00, A 0, B 0, C 0} C_DIS
LIN {X 91.84, Y 70.86, Z 0.00, A 0, B 0, C 0} C_DIS
LIN {X 91.93, Y 71.15, Z 0.00, A 0, B 0, C 0} C_DIS
LIN {X 92.03, Y 71.44, Z 0.00, A 0, B 0, C 0} C_DIS
LIN {X 92.14, Y 71.73, Z 0.00, A 0, B 0, C 0} C_DIS
LIN {X 92.24, Y 72.02, Z 0.00, A 0, B 0, C 0} C_DIS
LIN {X 92.34, Y 72.31, Z 0.00, A 0, B 0, C 0} C_DIS
LIN {X 92.45, Y 72.59, Z 0.00, A 0, B 0, C 0} C_DIS
LIN {X 92.55, Y 72.88, Z 0.00, A 0, B 0, C 0} C_DIS
LIN {X 92.66, Y 73.16, Z 0.00, A 0, B 0, C 0} C_DIS
LIN {X 92.77, Y 73.44, Z 0.00, A 0, B 0, C 0} C_DIS
LIN {X 92.88, Y 73.72, Z 0.00, A 0, B 0, C 0} C_DIS
LIN {X 92.99, Y 74.00, Z 0.00, A 0, B 0, C 0} C_DIS
LIN {X 93.11, Y 74.28, Z 0.00, A 0, B 0, C 0} C_DIS
LIN {X 93.23, Y 74.55, Z 0.00, A 0, B 0, C 0} C_DIS
LIN {X 93.35, Y 74.82, Z 0.00, A 0, B 0, C 0} C_DIS
LIN {X 93.48, Y 75.09, Z 0.00, A 0, B 0, C 0} C_DIS
LIN {X 93.61, Y 75.35, Z 0.00, A 0, B 0, C 0} C_DIS
LIN {X 93.74, Y 75.61, Z 0.00, A 0, B 0, C 0} C_DIS
LIN {X 93.88, Y 75.87, Z 0.00, A 0, B 0, C 0} C_DIS
LIN {X 94.01, Y 76.12, Z 0.00, A 0, B 0, C 0} C_DIS
LIN {X 94.16, Y 76.36, Z 0.00, A 0, B 0, C 0} C_DIS
LIN {X 94.30, Y 76.61, Z 0.00, A 0, B 0, C 0} C_DIS
LIN {X 94.45, Y 76.85, Z 0.00, A 0, B 0, C 0} C_DIS
LIN {X 94.60, Y 77.08, Z 0.00, A 0, B 0, C 0} C_DIS
LIN {X 94.75, Y 77.31, Z 0.00, A 0, B 0, C 0} C_DIS
LIN {X 94.91, Y 77.54, Z 0.00, A 0, B 0, C 0} C_DIS
LIN {X 95.07, Y 77.76, Z 0.00, A 0, B 0, C 0} C_DIS
LIN {X 95.22, Y 77.99, Z 0.00, A 0, B 0, C 0} C_DIS
LIN {X 95.38, Y 78.21, Z 0.00, A 0, B 0, C 0} C_DIS
LIN {X 95.54, Y 78.44, Z 0.00, A 0, B 0, C 0} C_DIS
LIN {X 95.69, Y 78.67, Z 0.00, A 0, B 0, C 0} C_DIS
LIN {X 95.85, Y 78.90, Z 0.00, A 0, B 0, C 0} C_DIS
LIN {X 96.00, Y 79.14, Z 0.00, A 0, B 0, C 0} C_DIS
LIN {X 96.15, Y 79.38, Z 0.00, A 0, B 0, C 0} C_DIS
LIN {X 96.30, Y 79.62, Z 0.00, A 0, B 0, C 0} C_DIS
LIN {X 96.45, Y 79.86, Z 0.00, A 0, B 0, C 0} C_DIS
LIN {X 96.60, Y 80.10, Z 0.00, A 0, B 0, C 0} C_DIS
LIN {X 96.75, Y 80.33, Z 0.00, A 0, B 0, C 0} C_DIS
LIN {X 96.91, Y 80.55, Z 0.00, A 0, B 0, C 0} C_DIS
LIN {X 97.07, Y 80.76, Z 0.00, A 0, B 0, C 0} C_DIS
LIN {X 97.24, Y 80.97, Z 0.00, A 0, B 0, C 0} C_DIS
LIN {X 97.42, Y 81.15, Z 0.00, A 0, B 0, C 0} C_DIS
LIN {X 97.60, Y 81.33, Z 0.00, A 0, B 0, C 0} C_DIS
LIN {X 97.78, Y 81.50, Z 0.00, A 0, B 0, C 0} C_DIS
LIN {X 97.97, Y 81.66, Z 0.00, A 0, B 0, C 0} C_DIS
LIN {X 98.16, Y 81.82, Z 0.00, A 0, B 0, C 0} C_DIS
LIN {X 98.36, Y 81.97, Z 0.00, A 0, B 0, C 0} C_DIS
LIN {X 98.55, Y 82.12, Z 0.00, A 0, B 0, C 0} C_DIS
LIN {X 98.74, Y 82.26, Z 0.00, A 0, B 0, C 0} C_DIS
LIN {X 98.94, Y 82.41, Z 0.00, A 0, B 0, C 0} C_DIS
LIN {X 99.13, Y 82.55, Z 0.00, A 0, B 0, C 0} C_DIS
LIN {X 99.33, Y 82.70, Z 0.00, A 0, B 0, C 0} C_DIS
LIN {X 99.52, Y 82.85, Z 0.00, A 0, B 0, C 0} C_DIS
LIN {X 99.71, Y 82.99, Z 0.00, A 0, B 0, C 0} C_DIS
LIN {X 99.91, Y 83.13, Z 0.00, A 0, B 0, C 0} C_DIS
LIN {X 100.10, Y 83.27, Z 0.00, A 0, B 0, C 0} C_DIS
LIN {X 100.29, Y 83.41, Z 0.00, A 0, B 0, C 0} C_DIS
LIN {X 100.49, Y 83.55, Z 0.00, A 0, B 0, C 0} C_DIS
LIN {X 100.69, Y 83.69, Z 0.00, A 0, B 0, C 0} C_DIS
LIN {X 100.88, Y 83.82, Z 0.00, A 0, B 0, C 0} C_DIS
LIN {X 101.08, Y 83.95, Z 0.00, A 0, B 0, C 0} C_DIS
LIN {X 101.29, Y 84.07, Z 0.00, A 0, B 0, C 0} C_DIS
LIN {X 101.49, Y 84.19, Z 0.00, A 0, B 0, C 0} C_DIS
LIN {X 101.69, Y 84.30, Z 0.00, A 0, B 0, C 0} C_DIS
LIN {X 101.90, Y 84.41, Z 0.00, A 0, B 0, C 0} C_DIS
LIN {X 102.11, Y 84.50, Z 0.00, A 0, B 0, C 0} C_DIS
LIN {X 102.32, Y 84.58, Z 0.00, A 0, B 0, C 0} C_DIS
LIN {X 102.53, Y 84.65, Z 0.00, A 0, B 0, C 0} C_DIS
LIN {X 102.74, Y 84.71, Z 0.00, A 0, B 0, C 0} C_DIS
LIN {X 102.96, Y 84.76, Z 0.00, A 0, B 0, C 0} C_DIS
LIN {X 103.17, Y 84.79, Z 0.00, A 0, B 0, C 0} C_DIS
LIN {X 103.39, Y 84.81, Z 0.00, A 0, B 0, C 0} C_DIS
LIN {X 103.60, Y 84.84, Z 0.00, A 0, B 0, C 0} C_DIS
LIN {X 103.82, Y 84.87, Z 0.00, A 0, B 0, C 0} C_DIS
LIN {X 104.03, Y 84.91, Z 0.00, A 0, B 0, C 0} C_DIS
LIN {X 104.25, Y 84.97, Z 0.00, A 0, B 0, C 0} C_DIS
LIN {X 104.46, Y 85.05, Z 0.00, A 0, B 0, C 0} C_DIS
LIN {X 104.67, Y 85.13, Z 0.00, A 0, B 0, C 0} C_DIS
LIN {X 104.88, Y 85.21, Z 0.00, A 0, B 0, C 0} C_DIS
LIN {X 105.09, Y 85.29, Z 0.00, A 0, B 0, C 0} C_DIS
LIN {X 105.30, Y 85.36, Z 0.00, A 0, B 0, C 0} C_DIS
LIN {X 105.52, Y 85.41, Z 0.00, A 0, B 0, C 0} C_DIS
LIN {X 105.73, Y 85.46, Z 0.00, A 0, B 0, C 0} C_DIS
LIN {X 105.95, Y 85.49, Z 0.00, A 0, B 0, C 0} C_DIS
LIN {X 106.16, Y 85.50, Z 0.00, A 0, B 0, C 0} C_DIS
LIN {X 106.38, Y 85.49, Z 0.00, A 0, B 0, C 0} C_DIS
LIN {X 106.59, Y 85.46, Z 0.00, A 0, B 0, C 0} C_DIS
LIN {X 106.81, Y 85.41, Z 0.00, A 0, B 0, C 0} C_DIS
LIN {X 107.02, Y 85.34, Z 0.00, A 0, B 0, C 0} C_DIS
LIN {X 107.24, Y 85.25, Z 0.00, A 0, B 0, C 0} C_DIS
LIN {X 107.24, Y 85.25, Z 10.00, A 0, B 0, C 0}

; ----- Contour 5 -----
PTP {X 163.01, Y 37.53, Z 10.00, A 0, B 0, C 0}
LIN {X 163.01, Y 37.53, Z 0.00, A 0, B 0, C 0}
LIN {X 162.79, Y 37.51, Z 0.00, A 0, B 0, C 0} C_DIS
LIN {X 162.58, Y 37.50, Z 0.00, A 0, B 0, C 0} C_DIS
LIN {X 162.36, Y 37.50, Z 0.00, A 0, B 0, C 0} C_DIS
LIN {X 162.15, Y 37.51, Z 0.00, A 0, B 0, C 0} C_DIS
LIN {X 161.93, Y 37.51, Z 0.00, A 0, B 0, C 0} C_DIS
LIN {X 161.71, Y 37.52, Z 0.00, A 0, B 0, C 0} C_DIS
LIN {X 161.49, Y 37.53, Z 0.00, A 0, B 0, C 0} C_DIS
LIN {X 161.27, Y 37.54, Z 0.00, A 0, B 0, C 0} C_DIS
LIN {X 161.05, Y 37.55, Z 0.00, A 0, B 0, C 0} C_DIS
LIN {X 160.84, Y 37.55, Z 0.00, A 0, B 0, C 0} C_DIS
LIN {X 160.62, Y 37.54, Z 0.00, A 0, B 0, C 0} C_DIS
LIN {X 160.40, Y 37.52, Z 0.00, A 0, B 0, C 0} C_DIS
LIN {X 160.19, Y 37.50, Z 0.00, A 0, B 0, C 0} C_DIS
LIN {X 159.98, Y 37.46, Z 0.00, A 0, B 0, C 0} C_DIS
LIN {X 159.76, Y 37.41, Z 0.00, A 0, B 0, C 0} C_DIS
LIN {X 159.55, Y 37.34, Z 0.00, A 0, B 0, C 0} C_DIS
LIN {X 159.35, Y 37.26, Z 0.00, A 0, B 0, C 0} C_DIS
LIN {X 159.14, Y 37.16, Z 0.00, A 0, B 0, C 0} C_DIS
LIN {X 158.94, Y 37.05, Z 0.00, A 0, B 0, C 0} C_DIS
LIN {X 158.74, Y 36.93, Z 0.00, A 0, B 0, C 0} C_DIS
LIN {X 158.54, Y 36.80, Z 0.00, A 0, B 0, C 0} C_DIS
LIN {X 158.35, Y 36.66, Z 0.00, A 0, B 0, C 0} C_DIS
LIN {X 158.16, Y 36.50, Z 0.00, A 0, B 0, C 0} C_DIS
LIN {X 157.97, Y 36.34, Z 0.00, A 0, B 0, C 0} C_DIS
LIN {X 157.78, Y 36.17, Z 0.00, A 0, B 0, C 0} C_DIS
LIN {X 157.60, Y 35.98, Z 0.00, A 0, B 0, C 0} C_DIS
LIN {X 157.42, Y 35.79, Z 0.00, A 0, B 0, C 0} C_DIS
LIN {X 157.25, Y 35.59, Z 0.00, A 0, B 0, C 0} C_DIS
LIN {X 157.08, Y 35.39, Z 0.00, A 0, B 0, C 0} C_DIS
LIN {X 156.92, Y 35.17, Z 0.00, A 0, B 0, C 0} C_DIS
LIN {X 156.76, Y 34.95, Z 0.00, A 0, B 0, C 0} C_DIS
LIN {X 156.61, Y 34.72, Z 0.00, A 0, B 0, C 0} C_DIS
LIN {X 156.46, Y 34.48, Z 0.00, A 0, B 0, C 0} C_DIS
LIN {X 156.31, Y 34.24, Z 0.00, A 0, B 0, C 0} C_DIS
LIN {X 156.17, Y 33.99, Z 0.00, A 0, B 0, C 0} C_DIS
LIN {X 156.04, Y 33.73, Z 0.00, A 0, B 0, C 0} C_DIS
LIN {X 155.91, Y 33.47, Z 0.00, A 0, B 0, C 0} C_DIS
LIN {X 155.79, Y 33.20, Z 0.00, A 0, B 0, C 0} C_DIS
LIN {X 155.68, Y 32.93, Z 0.00, A 0, B 0, C 0} C_DIS
LIN {X 155.57, Y 32.65, Z 0.00, A 0, B 0, C 0} C_DIS
LIN {X 155.46, Y 32.36, Z 0.00, A 0, B 0, C 0} C_DIS
LIN {X 155.37, Y 32.07, Z 0.00, A 0, B 0, C 0} C_DIS
LIN {X 155.28, Y 31.78, Z 0.00, A 0, B 0, C 0} C_DIS
LIN {X 155.20, Y 31.48, Z 0.00, A 0, B 0, C 0} C_DIS
LIN {X 155.12, Y 31.18, Z 0.00, A 0, B 0, C 0} C_DIS
LIN {X 155.05, Y 30.87, Z 0.00, A 0, B 0, C 0} C_DIS
LIN {X 154.99, Y 30.56, Z 0.00, A 0, B 0, C 0} C_DIS
LIN {X 154.94, Y 30.25, Z 0.00, A 0, B 0, C 0} C_DIS
LIN {X 154.90, Y 29.93, Z 0.00, A 0, B 0, C 0} C_DIS
LIN {X 154.86, Y 29.61, Z 0.00, A 0, B 0, C 0} C_DIS
LIN {X 154.83, Y 29.29, Z 0.00, A 0, B 0, C 0} C_DIS
LIN {X 154.81, Y 28.96, Z 0.00, A 0, B 0, C 0} C_DIS
LIN {X 154.79, Y 28.64, Z 0.00, A 0, B 0, C 0} C_DIS
LIN {X 154.78, Y 28.31, Z 0.00, A 0, B 0, C 0} C_DIS
LIN {X 154.78, Y 27.98, Z 0.00, A 0, B 0, C 0} C_DIS
LIN {X 154.78, Y 27.65, Z 0.00, A 0, B 0, C 0} C_DIS
LIN {X 154.79, Y 27.32, Z 0.00, A 0, B 0, C 0} C_DIS
LIN {X 154.80, Y 26.99, Z 0.00, A 0, B 0, C 0} C_DIS
LIN {X 154.82, Y 26.66, Z 0.00, A 0, B 0, C 0} C_DIS
LIN {X 154.84, Y 26.33, Z 0.00, A 0, B 0, C 0} C_DIS
LIN {X 154.86, Y 26.00, Z 0.00, A 0, B 0, C 0} C_DIS
LIN {X 154.90, Y 25.68, Z 0.00, A 0, B 0, C 0} C_DIS
LIN {X 154.93, Y 25.35, Z 0.00, A 0, B 0, C 0} C_DIS
LIN {X 154.97, Y 25.03, Z 0.00, A 0, B 0, C 0} C_DIS
LIN {X 155.01, Y 24.71, Z 0.00, A 0, B 0, C 0} C_DIS
LIN {X 155.07, Y 24.39, Z 0.00, A 0, B 0, C 0} C_DIS
LIN {X 155.12, Y 24.08, Z 0.00, A 0, B 0, C 0} C_DIS
LIN {X 155.19, Y 23.78, Z 0.00, A 0, B 0, C 0} C_DIS
LIN {X 155.26, Y 23.48, Z 0.00, A 0, B 0, C 0} C_DIS
LIN {X 155.34, Y 23.18, Z 0.00, A 0, B 0, C 0} C_DIS
LIN {X 155.44, Y 22.90, Z 0.00, A 0, B 0, C 0} C_DIS
LIN {X 155.54, Y 22.62, Z 0.00, A 0, B 0, C 0} C_DIS
LIN {X 155.65, Y 22.35, Z 0.00, A 0, B 0, C 0} C_DIS
LIN {X 155.78, Y 22.10, Z 0.00, A 0, B 0, C 0} C_DIS
LIN {X 155.92, Y 21.85, Z 0.00, A 0, B 0, C 0} C_DIS
LIN {X 156.07, Y 21.60, Z 0.00, A 0, B 0, C 0} C_DIS
LIN {X 156.22, Y 21.36, Z 0.00, A 0, B 0, C 0} C_DIS
LIN {X 156.38, Y 21.13, Z 0.00, A 0, B 0, C 0} C_DIS
LIN {X 156.53, Y 20.89, Z 0.00, A 0, B 0, C 0} C_DIS
LIN {X 156.69, Y 20.65, Z 0.00, A 0, B 0, C 0} C_DIS
LIN {X 156.84, Y 20.41, Z 0.00, A 0, B 0, C 0} C_DIS
LIN {X 156.99, Y 20.17, Z 0.00, A 0, B 0, C 0} C_DIS
LIN {X 157.15, Y 19.94, Z 0.00, A 0, B 0, C 0} C_DIS
LIN {X 157.31, Y 19.72, Z 0.00, A 0, B 0, C 0} C_DIS
LIN {X 157.48, Y 19.51, Z 0.00, A 0, B 0, C 0} C_DIS
LIN {X 157.65, Y 19.32, Z 0.00, A 0, B 0, C 0} C_DIS
LIN {X 157.83, Y 19.14, Z 0.00, A 0, B 0, C 0} C_DIS
LIN {X 158.01, Y 18.98, Z 0.00, A 0, B 0, C 0} C_DIS
LIN {X 158.20, Y 18.84, Z 0.00, A 0, B 0, C 0} C_DIS
LIN {X 158.39, Y 18.70, Z 0.00, A 0, B 0, C 0} C_DIS
LIN {X 158.59, Y 18.58, Z 0.00, A 0, B 0, C 0} C_DIS
LIN {X 158.79, Y 18.47, Z 0.00, A 0, B 0, C 0} C_DIS
LIN {X 158.99, Y 18.37, Z 0.00, A 0, B 0, C 0} C_DIS
LIN {X 159.20, Y 18.29, Z 0.00, A 0, B 0, C 0} C_DIS
LIN {X 159.41, Y 18.21, Z 0.00, A 0, B 0, C 0} C_DIS
LIN {X 159.62, Y 18.14, Z 0.00, A 0, B 0, C 0} C_DIS
LIN {X 159.83, Y 18.08, Z 0.00, A 0, B 0, C 0} C_DIS
LIN {X 160.05, Y 18.03, Z 0.00, A 0, B 0, C 0} C_DIS
LIN {X 160.26, Y 17.99, Z 0.00, A 0, B 0, C 0} C_DIS
LIN {X 160.48, Y 17.96, Z 0.00, A 0, B 0, C 0} C_DIS
LIN {X 160.70, Y 17.94, Z 0.00, A 0, B 0, C 0} C_DIS
LIN {X 160.92, Y 17.92, Z 0.00, A 0, B 0, C 0} C_DIS
LIN {X 161.14, Y 17.91, Z 0.00, A 0, B 0, C 0} C_DIS
LIN {X 161.36, Y 17.91, Z 0.00, A 0, B 0, C 0} C_DIS
LIN {X 161.58, Y 17.91, Z 0.00, A 0, B 0, C 0} C_DIS
LIN {X 161.79, Y 17.92, Z 0.00, A 0, B 0, C 0} C_DIS
LIN {X 162.01, Y 17.94, Z 0.00, A 0, B 0, C 0} C_DIS
LIN {X 162.23, Y 17.96, Z 0.00, A 0, B 0, C 0} C_DIS
LIN {X 162.45, Y 17.98, Z 0.00, A 0, B 0, C 0} C_DIS
LIN {X 162.66, Y 18.02, Z 0.00, A 0, B 0, C 0} C_DIS
LIN {X 162.88, Y 18.05, Z 0.00, A 0, B 0, C 0} C_DIS
LIN {X 163.09, Y 18.09, Z 0.00, A 0, B 0, C 0} C_DIS
LIN {X 163.30, Y 18.14, Z 0.00, A 0, B 0, C 0} C_DIS
LIN {X 163.51, Y 18.20, Z 0.00, A 0, B 0, C 0} C_DIS
LIN {X 163.71, Y 18.27, Z 0.00, A 0, B 0, C 0} C_DIS
LIN {X 163.92, Y 18.36, Z 0.00, A 0, B 0, C 0} C_DIS
LIN {X 164.12, Y 18.47, Z 0.00, A 0, B 0, C 0} C_DIS
LIN {X 164.32, Y 18.59, Z 0.00, A 0, B 0, C 0} C_DIS
LIN {X 164.51, Y 18.74, Z 0.00, A 0, B 0, C 0} C_DIS
LIN {X 164.70, Y 18.90, Z 0.00, A 0, B 0, C 0} C_DIS
LIN {X 164.89, Y 19.07, Z 0.00, A 0, B 0, C 0} C_DIS
LIN {X 165.07, Y 19.26, Z 0.00, A 0, B 0, C 0} C_DIS
LIN {X 165.25, Y 19.45, Z 0.00, A 0, B 0, C 0} C_DIS
LIN {X 165.42, Y 19.65, Z 0.00, A 0, B 0, C 0} C_DIS
LIN {X 165.59, Y 19.85, Z 0.00, A 0, B 0, C 0} C_DIS
LIN {X 165.75, Y 20.06, Z 0.00, A 0, B 0, C 0} C_DIS
LIN {X 165.91, Y 20.28, Z 0.00, A 0, B 0, C 0} C_DIS
LIN {X 166.07, Y 20.50, Z 0.00, A 0, B 0, C 0} C_DIS
LIN {X 166.22, Y 20.73, Z 0.00, A 0, B 0, C 0} C_DIS
LIN {X 166.36, Y 20.97, Z 0.00, A 0, B 0, C 0} C_DIS
LIN {X 166.51, Y 21.22, Z 0.00, A 0, B 0, C 0} C_DIS
LIN {X 166.64, Y 21.47, Z 0.00, A 0, B 0, C 0} C_DIS
LIN {X 166.77, Y 21.73, Z 0.00, A 0, B 0, C 0} C_DIS
LIN {X 166.90, Y 21.99, Z 0.00, A 0, B 0, C 0} C_DIS
LIN {X 167.02, Y 22.27, Z 0.00, A 0, B 0, C 0} C_DIS
LIN {X 167.14, Y 22.54, Z 0.00, A 0, B 0, C 0} C_DIS
LIN {X 167.24, Y 22.83, Z 0.00, A 0, B 0, C 0} C_DIS
LIN {X 167.34, Y 23.12, Z 0.00, A 0, B 0, C 0} C_DIS
LIN {X 167.44, Y 23.42, Z 0.00, A 0, B 0, C 0} C_DIS
LIN {X 167.52, Y 23.72, Z 0.00, A 0, B 0, C 0} C_DIS
LIN {X 167.59, Y 24.02, Z 0.00, A 0, B 0, C 0} C_DIS
LIN {X 167.66, Y 24.33, Z 0.00, A 0, B 0, C 0} C_DIS
LIN {X 167.71, Y 24.64, Z 0.00, A 0, B 0, C 0} C_DIS
LIN {X 167.75, Y 24.96, Z 0.00, A 0, B 0, C 0} C_DIS
LIN {X 167.78, Y 25.28, Z 0.00, A 0, B 0, C 0} C_DIS
LIN {X 167.80, Y 25.60, Z 0.00, A 0, B 0, C 0} C_DIS
LIN {X 167.81, Y 25.92, Z 0.00, A 0, B 0, C 0} C_DIS
LIN {X 167.81, Y 26.25, Z 0.00, A 0, B 0, C 0} C_DIS
LIN {X 167.81, Y 26.58, Z 0.00, A 0, B 0, C 0} C_DIS
LIN {X 167.81, Y 26.91, Z 0.00, A 0, B 0, C 0} C_DIS
LIN {X 167.81, Y 27.24, Z 0.00, A 0, B 0, C 0} C_DIS
LIN {X 167.80, Y 27.57, Z 0.00, A 0, B 0, C 0} C_DIS
LIN {X 167.80, Y 27.90, Z 0.00, A 0, B 0, C 0} C_DIS
LIN {X 167.80, Y 28.23, Z 0.00, A 0, B 0, C 0} C_DIS
LIN {X 167.80, Y 28.56, Z 0.00, A 0, B 0, C 0} C_DIS
LIN {X 167.80, Y 28.89, Z 0.00, A 0, B 0, C 0} C_DIS
LIN {X 167.79, Y 29.21, Z 0.00, A 0, B 0, C 0} C_DIS
LIN {X 167.77, Y 29.54, Z 0.00, A 0, B 0, C 0} C_DIS
LIN {X 167.75, Y 29.86, Z 0.00, A 0, B 0, C 0} C_DIS
LIN {X 167.72, Y 30.18, Z 0.00, A 0, B 0, C 0} C_DIS
LIN {X 167.69, Y 30.50, Z 0.00, A 0, B 0, C 0} C_DIS
LIN {X 167.64, Y 30.82, Z 0.00, A 0, B 0, C 0} C_DIS
LIN {X 167.58, Y 31.13, Z 0.00, A 0, B 0, C 0} C_DIS
LIN {X 167.52, Y 31.44, Z 0.00, A 0, B 0, C 0} C_DIS
LIN {X 167.44, Y 31.75, Z 0.00, A 0, B 0, C 0} C_DIS
LIN {X 167.36, Y 32.04, Z 0.00, A 0, B 0, C 0} C_DIS
LIN {X 167.27, Y 32.34, Z 0.00, A 0, B 0, C 0} C_DIS
LIN {X 167.17, Y 32.63, Z 0.00, A 0, B 0, C 0} C_DIS
LIN {X 167.06, Y 32.91, Z 0.00, A 0, B 0, C 0} C_DIS
LIN {X 166.94, Y 33.18, Z 0.00, A 0, B 0, C 0} C_DIS
LIN {X 166.82, Y 33.45, Z 0.00, A 0, B 0, C 0} C_DIS
LIN {X 166.69, Y 33.70, Z 0.00, A 0, B 0, C 0} C_DIS
LIN {X 166.55, Y 33.96, Z 0.00, A 0, B 0, C 0} C_DIS
LIN {X 166.40, Y 34.20, Z 0.00, A 0, B 0, C 0} C_DIS
LIN {X 166.25, Y 34.44, Z 0.00, A 0, B 0, C 0} C_DIS
LIN {X 166.10, Y 34.66, Z 0.00, A 0, B 0, C 0} C_DIS
LIN {X 165.94, Y 34.89, Z 0.00, A 0, B 0, C 0} C_DIS
LIN {X 165.77, Y 35.10, Z 0.00, A 0, B 0, C 0} C_DIS
LIN {X 165.60, Y 35.31, Z 0.00, A 0, B 0, C 0} C_DIS
LIN {X 165.43, Y 35.51, Z 0.00, A 0, B 0, C 0} C_DIS
LIN {X 165.25, Y 35.70, Z 0.00, A 0, B 0, C 0} C_DIS
LIN {X 165.08, Y 35.89, Z 0.00, A 0, B 0, C 0} C_DIS
LIN {X 164.90, Y 36.07, Z 0.00, A 0, B 0, C 0} C_DIS
LIN {X 164.72, Y 36.24, Z 0.00, A 0, B 0, C 0} C_DIS
LIN {X 164.54, Y 36.41, Z 0.00, A 0, B 0, C 0} C_DIS
LIN {X 164.35, Y 36.57, Z 0.00, A 0, B 0, C 0} C_DIS
LIN {X 164.16, Y 36.73, Z 0.00, A 0, B 0, C 0} C_DIS
LIN {X 163.97, Y 36.88, Z 0.00, A 0, B 0, C 0} C_DIS
LIN {X 163.78, Y 37.03, Z 0.00, A 0, B 0, C 0} C_DIS
LIN {X 163.59, Y 37.18, Z 0.00, A 0, B 0, C 0} C_DIS
LIN {X 163.39, Y 37.32, Z 0.00, A 0, B 0, C 0} C_DIS
LIN {X 163.39, Y 37.32, Z 10.00, A 0, B 0, C 0}

; ----- Contour 6 -----
PTP {X 163.24, Y 36.45, Z 10.00, A 0, B 0, C 0}
LIN {X 163.24, Y 36.45, Z 0.00, A 0, B 0, C 0}
LIN {X 163.44, Y 36.34, Z 0.00, A 0, B 0, C 0} C_DIS
LIN {X 163.64, Y 36.22, Z 0.00, A 0, B 0, C 0} C_DIS
LIN {X 163.84, Y 36.09, Z 0.00, A 0, B 0, C 0} C_DIS
LIN {X 164.04, Y 35.94, Z 0.00, A 0, B 0, C 0} C_DIS
LIN {X 164.23, Y 35.79, Z 0.00, A 0, B 0, C 0} C_DIS
LIN {X 164.41, Y 35.62, Z 0.00, A 0, B 0, C 0} C_DIS
LIN {X 164.60, Y 35.45, Z 0.00, A 0, B 0, C 0} C_DIS
LIN {X 164.77, Y 35.26, Z 0.00, A 0, B 0, C 0} C_DIS
LIN {X 164.95, Y 35.07, Z 0.00, A 0, B 0, C 0} C_DIS
LIN {X 165.12, Y 34.86, Z 0.00, A 0, B 0, C 0} C_DIS
LIN {X 165.28, Y 34.65, Z 0.00, A 0, B 0, C 0} C_DIS
LIN {X 165.44, Y 34.43, Z 0.00, A 0, B 0, C 0} C_DIS
LIN {X 165.60, Y 34.20, Z 0.00, A 0, B 0, C 0} C_DIS
LIN {X 165.75, Y 33.97, Z 0.00, A 0, B 0, C 0} C_DIS
LIN {X 165.90, Y 33.72, Z 0.00, A 0, B 0, C 0} C_DIS
LIN {X 166.04, Y 33.47, Z 0.00, A 0, B 0, C 0} C_DIS
LIN {X 166.17, Y 33.21, Z 0.00, A 0, B 0, C 0} C_DIS
LIN {X 166.30, Y 32.95, Z 0.00, A 0, B 0, C 0} C_DIS
LIN {X 166.42, Y 32.68, Z 0.00, A 0, B 0, C 0} C_DIS
LIN {X 166.54, Y 32.40, Z 0.00, A 0, B 0, C 0} C_DIS
LIN {X 166.65, Y 32.12, Z 0.00, A 0, B 0, C 0} C_DIS
LIN {X 166.76, Y 31.84, Z 0.00, A 0, B 0, C 0} C_DIS
LIN {X 166.85, Y 31.54, Z 0.00, A 0, B 0, C 0} C_DIS
LIN {X 166.95, Y 31.25, Z 0.00, A 0, B 0, C 0} C_DIS
LIN {X 167.03, Y 30.95, Z 0.00, A 0, B 0, C 0} C_DIS
LIN {X 167.11, Y 30.65, Z 0.00, A 0, B 0, C 0} C_DIS
LIN {X 167.18, Y 30.34, Z 0.00, A 0, B 0, C 0} C_DIS
LIN {X 167.24, Y 30.03, Z 0.00, A 0, B 0, C 0} C_DIS
LIN {X 167.30, Y 29.72, Z 0.00, A 0, B 0, C 0} C_DIS
LIN {X 167.35, Y 29.41, Z 0.00, A 0, B 0, C 0} C_DIS
LIN {X 167.39, Y 29.09, Z 0.00, A 0, B 0, C 0} C_DIS
LIN {X 167.42, Y 28.77, Z 0.00, A 0, B 0, C 0} C_DIS
LIN {X 167.45, Y 28.45, Z 0.00, A 0, B 0, C 0} C_DIS
LIN {X 167.47, Y 28.13, Z 0.00, A 0, B 0, C 0} C_DIS
LIN {X 167.47, Y 27.81, Z 0.00, A 0, B 0, C 0} C_DIS
LIN {X 167.48, Y 27.49, Z 0.00, A 0, B 0, C 0} C_DIS
LIN {X 167.47, Y 27.17, Z 0.00, A 0, B 0, C 0} C_DIS
LIN {X 167.45, Y 26.85, Z 0.00, A 0, B 0, C 0} C_DIS
LIN {X 167.42, Y 26.53, Z 0.00, A 0, B 0, C 0} C_DIS
LIN {X 167.39, Y 26.21, Z 0.00, A 0, B 0, C 0} C_DIS
LIN {X 167.35, Y 25.89, Z 0.00, A 0, B 0, C 0} C_DIS
LIN {X 167.29, Y 25.57, Z 0.00, A 0, B 0, C 0} C_DIS
LIN {X 167.23, Y 25.26, Z 0.00, A 0, B 0, C 0} C_DIS
LIN {X 167.16, Y 24.95, Z 0.00, A 0, B 0, C 0} C_DIS
LIN {X 167.07, Y 24.64, Z 0.00, A 0, B 0, C 0} C_DIS
LIN {X 166.99, Y 24.33, Z 0.00, A 0, B 0, C 0} C_DIS
LIN {X 166.89, Y 24.03, Z 0.00, A 0, B 0, C 0} C_DIS
LIN {X 166.79, Y 23.72, Z 0.00, A 0, B 0, C 0} C_DIS
LIN {X 166.70, Y 23.42, Z 0.00, A 0, B 0, C 0} C_DIS
LIN {X 166.60, Y 23.13, Z 0.00, A 0, B 0, C 0} C_DIS
LIN {X 166.49, Y 22.83, Z 0.00, A 0, B 0, C 0} C_DIS
LIN {X 166.39, Y 22.54, Z 0.00, A 0, B 0, C 0} C_DIS
LIN {X 166.28, Y 22.26, Z 0.00, A 0, B 0, C 0} C_DIS
LIN {X 166.17, Y 21.99, Z 0.00, A 0, B 0, C 0} C_DIS
LIN {X 166.05, Y 21.73, Z 0.00, A 0, B 0, C 0} C_DIS
LIN {X 165.92, Y 21.48, Z 0.00, A 0, B 0, C 0} C_DIS
LIN {X 165.79, Y 21.25, Z 0.00, A 0, B 0, C 0} C_DIS
LIN {X 165.64, Y 21.02, Z 0.00, A 0, B 0, C 0} C_DIS
LIN {X 165.49, Y 20.82, Z 0.00, A 0, B 0, C 0} C_DIS
LIN {X 165.32, Y 20.62, Z 0.00, A 0, B 0, C 0} C_DIS
LIN {X 165.15, Y 20.44, Z 0.00, A 0, B 0, C 0} C_DIS
LIN {X 164.97, Y 20.27, Z 0.00, A 0, B 0, C 0} C_DIS
LIN {X 164.78, Y 20.11, Z 0.00, A 0, B 0, C 0} C_DIS
LIN {X 164.59, Y 19.95, Z 0.00, A 0, B 0, C 0} C_DIS
LIN {X 164.39, Y 19.80, Z 0.00, A 0, B 0, C 0} C_DIS
LIN {X 164.20, Y 19.64, Z 0.00, A 0, B 0, C 0} C_DIS
LIN {X 164.00, Y 19.50, Z 0.00, A 0, B 0, C 0} C_DIS
LIN {X 163.80, Y 19.36, Z 0.00, A 0, B 0, C 0} C_DIS
LIN {X 163.60, Y 19.22, Z 0.00, A 0, B 0, C 0} C_DIS
LIN {X 163.40, Y 19.09, Z 0.00, A 0, B 0, C 0} C_DIS
LIN {X 163.19, Y 18.98, Z 0.00, A 0, B 0, C 0} C_DIS
LIN {X 162.99, Y 18.87, Z 0.00, A 0, B 0, C 0} C_DIS
LIN {X 162.78, Y 18.77, Z 0.00, A 0, B 0, C 0} C_DIS
LIN {X 162.57, Y 18.68, Z 0.00, A 0, B 0, C 0} C_DIS
LIN {X 162.36, Y 18.61, Z 0.00, A 0, B 0, C 0} C_DIS
LIN {X 162.15, Y 18.55, Z 0.00, A 0, B 0, C 0} C_DIS
LIN {X 161.94, Y 18.51, Z 0.00, A 0, B 0, C 0} C_DIS
LIN {X 161.72, Y 18.48, Z 0.00, A 0, B 0, C 0} C_DIS
LIN {X 161.51, Y 18.47, Z 0.00, A 0, B 0, C 0} C_DIS
LIN {X 161.30, Y 18.47, Z 0.00, A 0, B 0, C 0} C_DIS
LIN {X 161.08, Y 18.48, Z 0.00, A 0, B 0, C 0} C_DIS
LIN {X 160.87, Y 18.50, Z 0.00, A 0, B 0, C 0} C_DIS
LIN {X 160.66, Y 18.54, Z 0.00, A 0, B 0, C 0} C_DIS
LIN {X 160.45, Y 18.59, Z 0.00, A 0, B 0, C 0} C_DIS
LIN {X 160.24, Y 18.65, Z 0.00, A 0, B 0, C 0} C_DIS
LIN {X 160.03, Y 18.72, Z 0.00, A 0, B 0, C 0} C_DIS
LIN {X 159.82, Y 18.80, Z 0.00, A 0, B 0, C 0} C_DIS
LIN {X 159.61, Y 18.90, Z 0.00, A 0, B 0, C 0} C_DIS
LIN {X 159.41, Y 19.01, Z 0.00, A 0, B 0, C 0} C_DIS
LIN {X 159.21, Y 19.12, Z 0.00, A 0, B 0, C 0} C_DIS
LIN {X 159.01, Y 19.25, Z 0.00, A 0, B 0, C 0} C_DIS
LIN {X 158.81, Y 19.39, Z 0.00, A 0, B 0, C 0} C_DIS
LIN {X 158.62, Y 19.54, Z 0.00, A 0, B 0, C 0} C_DIS
LIN {X 158.42, Y 19.69, Z 0.00, A 0, B 0, C 0} C_DIS
LIN {X 158.24, Y 19.86, Z 0.00, A 0, B 0, C 0} C_DIS
LIN {X 158.05, Y 20.04, Z 0.00, A 0, B 0, C 0} C_DIS
LIN {X 157.87, Y 20.22, Z 0.00, A 0, B 0, C 0} C_DIS
LIN {X 157.70, Y 20.41, Z 0.00, A 0, B 0, C 0} C_DIS
LIN {X 157.52, Y 20.62, Z 0.00, A 0, B 0, C 0} C_DIS
LIN {X 157.36, Y 20.83, Z 0.00, A 0, B 0, C 0} C_DIS
LIN {X 157.19, Y 21.05, Z 0.00, A 0, B 0, C 0} C_DIS
LIN {X 157.04, Y 21.27, Z 0.00, A 0, B 0, C 0} C_DIS
LIN {X 156.88, Y 21.51, Z 0.00, A 0, B 0, C 0} C_DIS
LIN {X 156.74, Y 21.75, Z 0.00, A 0, B 0, C 0} C_DIS
LIN {X 156.59, Y 22.00, Z 0.00, A 0, B 0, C 0} C_DIS
LIN {X 156.46, Y 22.25, Z 0.00, A 0, B 0, C 0} C_DIS
LIN {X 156.33, Y 22.52, Z 0.00, A 0, B 0, C 0} C_DIS
LIN {X 156.21, Y 22.78, Z 0.00, A 0, B 0, C 0} C_DIS
LIN {X 156.09, Y 23.06, Z 0.00, A 0, B 0, C 0} C_DIS
LIN {X 155.98, Y 23.34, Z 0.00, A 0, B 0, C 0} C_DIS
LIN {X 155.87, Y 23.63, Z 0.00, A 0, B 0, C 0} C_DIS
LIN {X 155.78, Y 23.92, Z 0.00, A 0, B 0, C 0} C_DIS
LIN {X 155.69, Y 24.22, Z 0.00, A 0, B 0, C 0} C_DIS
LIN {X 155.60, Y 24.52, Z 0.00, A 0, B 0, C 0} C_DIS
LIN {X 155.53, Y 24.82, Z 0.00, A 0, B 0, C 0} C_DIS
LIN {X 155.46, Y 25.13, Z 0.00, A 0, B 0, C 0} C_DIS
LIN {X 155.40, Y 25.44, Z 0.00, A 0, B 0, C 0} C_DIS
LIN {X 155.34, Y 25.75, Z 0.00, A 0, B 0, C 0} C_DIS
LIN {X 155.30, Y 26.07, Z 0.00, A 0, B 0, C 0} C_DIS
LIN {X 155.26, Y 26.39, Z 0.00, A 0, B 0, C 0} C_DIS
LIN {X 155.23, Y 26.71, Z 0.00, A 0, B 0, C 0} C_DIS
LIN {X 155.20, Y 27.03, Z 0.00, A 0, B 0, C 0} C_DIS
LIN {X 155.19, Y 27.35, Z 0.00, A 0, B 0, C 0} C_DIS
LIN {X 155.18, Y 27.68, Z 0.00, A 0, B 0, C 0} C_DIS
LIN {X 155.18, Y 28.00, Z 0.00, A 0, B 0, C 0} C_DIS
LIN {X 155.18, Y 28.32, Z 0.00, A 0, B 0, C 0} C_DIS
LIN {X 155.20, Y 28.64, Z 0.00, A 0, B 0, C 0} C_DIS
LIN {X 155.22, Y 28.96, Z 0.00, A 0, B 0, C 0} C_DIS
LIN {X 155.25, Y 29.28, Z 0.00, A 0, B 0, C 0} C_DIS
LIN {X 155.29, Y 29.60, Z 0.00, A 0, B 0, C 0} C_DIS
LIN {X 155.34, Y 29.91, Z 0.00, A 0, B 0, C 0} C_DIS
LIN {X 155.40, Y 30.22, Z 0.00, A 0, B 0, C 0} C_DIS
LIN {X 155.46, Y 30.53, Z 0.00, A 0, B 0, C 0} C_DIS
LIN {X 155.54, Y 30.83, Z 0.00, A 0, B 0, C 0} C_DIS
LIN {X 155.62, Y 31.13, Z 0.00, A 0, B 0, C 0} C_DIS
LIN {X 155.71, Y 31.43, Z 0.00, A 0, B 0, C 0} C_DIS
LIN {X 155.80, Y 31.72, Z 0.00, A 0, B 0, C 0} C_DIS
LIN {X 155.91, Y 32.01, Z 0.00, A 0, B 0, C 0} C_DIS
LIN {X 156.02, Y 32.29, Z 0.00, A 0, B 0, C 0} C_DIS
LIN {X 156.14, Y 32.57, Z 0.00, A 0, B 0, C 0} C_DIS
LIN {X 156.26, Y 32.84, Z 0.00, A 0, B 0, C 0} C_DIS
LIN {X 156.39, Y 33.10, Z 0.00, A 0, B 0, C 0} C_DIS
LIN {X 156.53, Y 33.36, Z 0.00, A 0, B 0, C 0} C_DIS
LIN {X 156.67, Y 33.62, Z 0.00, A 0, B 0, C 0} C_DIS
LIN {X 156.82, Y 33.86, Z 0.00, A 0, B 0, C 0} C_DIS
LIN {X 156.97, Y 34.10, Z 0.00, A 0, B 0, C 0} C_DIS
LIN {X 157.13, Y 34.33, Z 0.00, A 0, B 0, C 0} C_DIS
LIN {X 157.29, Y 34.56, Z 0.00, A 0, B 0, C 0} C_DIS
LIN {X 157.46, Y 34.77, Z 0.00, A 0, B 0, C 0} C_DIS
LIN {X 157.63, Y 34.98, Z 0.00, A 0, B 0, C 0} C_DIS
LIN {X 157.80, Y 35.18, Z 0.00, A 0, B 0, C 0} C_DIS
LIN {X 157.98, Y 35.37, Z 0.00, A 0, B 0, C 0} C_DIS
LIN {X 158.16, Y 35.55, Z 0.00, A 0, B 0, C 0} C_DIS
LIN {X 158.34, Y 35.73, Z 0.00, A 0, B 0, C 0} C_DIS
LIN {X 158.53, Y 35.89, Z 0.00, A 0, B 0, C 0} C_DIS
LIN {X 158.72, Y 36.04, Z 0.00, A 0, B 0, C 0} C_DIS
LIN {X 158.91, Y 36.19, Z 0.00, A 0, B 0, C 0} C_DIS
LIN {X 159.10, Y 36.32, Z 0.00, A 0, B 0, C 0} C_DIS
LIN {X 159.30, Y 36.44, Z 0.00, A 0, B 0, C 0} C_DIS
LIN {X 159.50, Y 36.55, Z 0.00, A 0, B 0, C 0} C_DIS
LIN {X 159.70, Y 36.65, Z 0.00, A 0, B 0, C 0} C_DIS
LIN {X 159.90, Y 36.74, Z 0.00, A 0, B 0, C 0} C_DIS
LIN {X 160.11, Y 36.82, Z 0.00, A 0, B 0, C 0} C_DIS
LIN {X 160.32, Y 36.89, Z 0.00, A 0, B 0, C 0} C_DIS
LIN {X 160.53, Y 36.95, Z 0.00, A 0, B 0, C 0} C_DIS
LIN {X 160.74, Y 36.99, Z 0.00, A 0, B 0, C 0} C_DIS
LIN {X 160.95, Y 37.02, Z 0.00, A 0, B 0, C 0} C_DIS
LIN {X 161.17, Y 37.04, Z 0.00, A 0, B 0, C 0} C_DIS
LIN {X 161.38, Y 37.05, Z 0.00, A 0, B 0, C 0} C_DIS
LIN {X 161.60, Y 37.04, Z 0.00, A 0, B 0, C 0} C_DIS
LIN {X 161.82, Y 37.02, Z 0.00, A 0, B 0, C 0} C_DIS
LIN {X 162.04, Y 36.99, Z 0.00, A 0, B 0, C 0} C_DIS
LIN {X 162.26, Y 36.95, Z 0.00, A 0, B 0, C 0} C_DIS
LIN {X 162.48, Y 36.89, Z 0.00, A 0, B 0, C 0} C_DIS
LIN {X 162.70, Y 36.82, Z 0.00, A 0, B 0, C 0} C_DIS
LIN {X 162.93, Y 36.74, Z 0.00, A 0, B 0, C 0} C_DIS
LIN {X 162.93, Y 36.74, Z 10.00, A 0, B 0, C 0}

